LIN {X 0,Y 131.785,Z 325.121,A -85,B 0,C 180,E1 -26219.114,E2 -26219.114} C_VEL
LIN {X 0,Y 136.517,Z 312.595,A -85,B 0,C 180,E1 -26221.843,E2 -26221.843} C_VEL
LIN {X 0,Y 140.644,Z 299.524,A -85,B 0,C 180,E1 -26223.984,E2 -26223.984} C_VEL
LIN {X 0,Y 143.918,Z 286.061,A -85,B 0,C 180,E1 -26225.653,E2 -26225.653} C_VEL
LIN {X 0,Y 146.479,Z 272.18,A -85,B 0,C 180,E1 -26226.846,E2 -26226.846} C_VEL
LIN {X 0,Y 148.119,Z 259.286,A -85,B 0,C 180,E1 -26227.542,E2 -26227.542} C_VEL
LIN {X 0,Y 152.361,Z 207.8,A -85,B 0,C 180,E1 -26229.457,E2 -26229.457} C_VEL
LIN {X 0,Y 147.363,Z 196.9,A -85,B 0,C 180,E1 -26232.578,E2 -26232.578} C_VEL
LIN {X 0,Y 142.317,Z 187.434,A -85,B 0,C 180,E1 -26236.042,E2 -26236.042} C_VEL
LIN {X 0,Y 138.298,Z 180.817,A -85,B 0,C 180,E1 -26239.137,E2 -26239.137} C_VEL
LIN {X 0,Y 134.118,Z 174.322,A -85,B 0,C 180,E1 -26242.853,E2 -26242.853} C_VEL
LIN {X 0,Y 130.981,Z 169.962,A -85,B 0,C 180,E1 -26246.076,E2 -26246.076} C_VEL
LIN {X 0,Y 128.411,Z 166.477,A -85,B 0,C 180,E1 -26249.154,E2 -26249.154} C_VEL
LIN {X 0,Y 127.763,Z 165.521,A -85,B 0,C 180,E1 -26250.031,E2 -26250.031} C_VEL
LIN {X 0,Y 125.309,Z 162.834,A -85,B 0,C 180,E1 -26253.6,E2 -26253.6} C_VEL
LIN {X 0,Y 124.174,Z 160.568,A -85,B 0,C 180,E1 -26255.787,E2 -26255.787} C_VEL
LIN {X 0,Y 121.255,Z 158.023,A -85,B 0,C 180,E1 -26262.732,E2 -26262.732} C_VEL
LIN {X 0,Y 120.363,Z 155.046,A -85,B 0,C 180,E1 -26268.375,E2 -26268.375} C_VEL
LIN {X 0,Y 120.599,Z 154.855,A -85,B 0,C 180,E1 -26276.67,E2 -26276.67} C_VEL
LIN {X 0,Y 120.863,Z 155.058,A -85,B 0,C 180,E1 -26278.137,E2 -26278.137} C_VEL
LIN {X 0,Y 121.622,Z 157.801,A -85,B 0,C 180,E1 -26281.874,E2 -26281.874} C_VEL
LIN {X 0,Y 123.928,Z 160.174,A -85,B 0,C 180,E1 -26287.341,E2 -26287.341} C_VEL
LIN {X 0,Y 124.584,Z 160.744,A -85,B 0,C 180,E1 -26288.526,E2 -26288.526} C_VEL
LIN {X 0,Y 126.362,Z 163.972,A -85,B 0,C 180,E1 -26291.642,E2 -26291.642} C_VEL
LIN {X 0,Y 128.449,Z 166.176,A -85,B 0,C 180,E1 -26294.466,E2 -26294.466} C_VEL
LIN {X 0,Y 131.151,Z 169.964,A -85,B 0,C 180,E1 -26297.718,E2 -26297.718} C_VEL
LIN {X 0,Y 135.213,Z 176.102,A -85,B 0,C 180,E1 -26301.831,E2 -26301.831} C_VEL
LIN {X 0,Y 137.802,Z 180.05,A -85,B 0,C 180,E1 -26304.089,E2 -26304.089} C_VEL
LIN {X 0,Y 142.126,Z 187.185,A -85,B 0,C 180,E1 -26307.455,E2 -26307.455} C_VEL
LIN {X 0,Y 145.883,Z 194.238,A -85,B 0,C 180,E1 -26310.095,E2 -26310.095} C_VEL
LIN {X 0,Y 150.285,Z 206.436,A -85,B 0,C 180,E1 -26313.156,E2 -26313.156} C_VEL
LIN {X 0,Y 152.14,Z 212.6,A -85,B 0,C 180,E1 -26314.415,E2 -26314.415} C_VEL
LIN {X 0,Y 147.502,Z 269.5,A -85,B 0,C 180,E1 -26316.633,E2 -26316.633} C_VEL
LIN {X 0,Y 145.233,Z 284.149,A -85,B 0,C 180,E1 -26317.596,E2 -26317.596} C_VEL
LIN {X 0,Y 142.182,Z 297.577,A -85,B 0,C 180,E1 -26318.882,E2 -26318.882} C_VEL
LIN {X 0,Y 138.14,Z 311.67,A -85,B 0,C 180,E1 -26320.826,E2 -26320.826} C_VEL
LIN {X 0,Y 133.661,Z 324.178,A -85,B 0,C 180,E1 -26323.133,E2 -26323.133} C_VEL
LIN {X 0,Y 130.05,Z 333.38,A -85,B 0,C 180,E1 -26325.376,E2 -26325.376} C_VEL
LIN {X 0,Y 126.93,Z 340.175,A -85,B 0,C 180,E1 -26327.298,E2 -26327.298} C_VEL
LIN {X 0,Y 122.296,Z 349.988,A -85,B 0,C 180,E1 -26330.798,E2 -26330.798} C_VEL
LIN {X 0,Y 117.358,Z 359.79,A -85,B 0,C 180,E1 -26335.332,E2 -26335.332} C_VEL
LIN {X 0,Y 112.94,Z 368.47,A -85,B 0,C 180,E1 -26340.617,E2 -26340.617} C_VEL
LIN {X 0,Y 109.945,Z 374.628,A -85,B 0,C 180,E1 -26345.455,E2 -26345.455} C_VEL
LIN {X 0,Y 107.473,Z 380.188,A -85,B 0,C 180,E1 -26350.921,E2 -26350.921} C_VEL
LIN {X 0,Y 105.927,Z 384.738,A -85,B 0,C 180,E1 -26356.578,E2 -26356.578} C_VEL
LIN {X 0,Y 105.224,Z 388.285,A -85,B 0,C 180,E1 -26362.329,E2 -26362.329} C_VEL
LIN {X 0,Y 105.192,Z 391.7,A -85,B 0,C 180,E1 -26370.005,E2 -26370.005} C_VEL
LIN {X 0,Y 105.119,Z 392.843,A -85,B 0,C 180,E1 -26373.839,E2 -26373.839} C_VEL
LIN {X 0,Y 105.704,Z 394.109,A -85,B 0,C 180,E1 -26381.511,E2 -26381.511} C_VEL
LIN {X 0,Y 107.789,Z 394.075,A -85,B 0,C 180,E1 -26389.032,E2 -26389.032} C_VEL
LIN {X 0,Y 111.681,Z 392.762,A -85,B 0,C 180,E1 -26396.141,E2 -26396.141} C_VEL
LIN {X 0,Y 117.55,Z 389.878,A -85,B 0,C 180,E1 -26403.156,E2 -26403.156} C_VEL
LIN {X 0,Y 124.609,Z 385.666,A -85,B 0,C 180,E1 -26409.134,E2 -26409.134} C_VEL
LIN {X 0,Y 127.112,Z 383.711,A -85,B 0,C 180,E1 -26411.401,E2 -26411.401} C_VEL
LIN {X 0,Y 130.13,Z 380.239,A -85,B 0,C 180,E1 -26415.327,E2 -26415.327} C_VEL
LIN {X 0,Y 133.647,Z 376.305,A -85,B 0,C 180,E1 -26418.958,E2 -26418.958} C_VEL
LIN {X 0,Y 136.798,Z 373.53,A -85,B 0,C 180,E1 -26420.711,E2 -26420.711} C_VEL
LIN {X 0,Y 145.544,Z 366.023,A -85,B 0,C 180,E1 -26423.987,E2 -26423.987} C_VEL
LIN {X 0,Y 154.63,Z 356.799,A -85,B 0,C 180,E1 -26426.995,E2 -26426.995} C_VEL
LIN {X 0,Y 163.45,Z 346.525,A -85,B 0,C 180,E1 -26429.318,E2 -26429.318} C_VEL
LIN {X 0,Y 171.421,Z 335.451,A -85,B 0,C 180,E1 -26431.211,E2 -26431.211} C_VEL
LIN {X 0,Y 178.854,Z 323.08,A -85,B 0,C 180,E1 -26432.759,E2 -26432.759} C_VEL
LIN {X 0,Y 184.948,Z 310.841,A -85,B 0,C 180,E1 -26433.87,E2 -26433.87} C_VEL
LIN {X 0,Y 190.356,Z 297.238,A -85,B 0,C 180,E1 -26434.769,E2 -26434.769} C_VEL
LIN {X 0,Y 194.439,Z 283.649,A -85,B 0,C 180,E1 -26435.428,E2 -26435.428} C_VEL
LIN {X 0,Y 197.393,Z 269.461,A -85,B 0,C 180,E1 -26435.918,E2 -26435.918} C_VEL
LIN {X 0,Y 199.287,Z 253.75,A -85,B 0,C 180,E1 -26436.344,E2 -26436.344} C_VEL
LIN {X 0,Y 197.239,Z 247.184,A -85,B 0,C 180,E1 -26439.469,E2 -26439.469} C_VEL
LIN {X 0,Y 195.601,Z 242.329,A -85,B 0,C 180,E1 -26442.751,E2 -26442.751} C_VEL
LIN {X 0,Y 194.612,Z 239.828,A -85,B 0,C 180,E1 -26445.351,E2 -26445.351} C_VEL
LIN {X 0,Y 193.533,Z 236.708,A -85,B 0,C 180,E1 -26451.641,E2 -26451.641} C_VEL
LIN {X 0,Y 193.655,Z 236.699,A -85,B 0,C 180,E1 -26454.175,E2 -26454.175} C_VEL
LIN {X 0,Y 194.972,Z 240.283,A -85,B 0,C 180,E1 -26459.993,E2 -26459.993} C_VEL
LIN {X 0,Y 196.407,Z 243.777,A -85,B 0,C 180,E1 -26463.231,E2 -26463.231} C_VEL
LIN {X 0,Y 198.462,Z 248.413,A -85,B 0,C 180,E1 -26466.533,E2 -26466.533} C_VEL
LIN {X 0,Y 199.581,Z 251.089,A -85,B 0,C 180,E1 -26468.026,E2 -26468.026} C_VEL
LIN {X 0,Y 197.317,Z 268.586,A -85,B 0,C 180,E1 -26468.483,E2 -26468.483} C_VEL
LIN {X 0,Y 194.205,Z 282.706,A -85,B 0,C 180,E1 -26469.03,E2 -26469.03} C_VEL
LIN {X 0,Y 190.296,Z 295.309,A -85,B 0,C 180,E1 -26469.712,E2 -26469.712} C_VEL
LIN {X 0,Y 185.117,Z 308.406,A -85,B 0,C 180,E1 -26470.741,E2 -26470.741} C_VEL
LIN {X 0,Y 178.785,Z 321.148,A -85,B 0,C 180,E1 -26472.074,E2 -26472.074} C_VEL
LIN {X 0,Y 171.815,Z 332.614,A -85,B 0,C 180,E1 -26473.649,E2 -26473.649} C_VEL
LIN {X 0,Y 164.146,Z 343.198,A -85,B 0,C 180,E1 -26475.548,E2 -26475.548} C_VEL
LIN {X 0,Y 156.73,Z 352.032,A -85,B 0,C 180,E1 -26477.648,E2 -26477.648} C_VEL
LIN {X 0,Y 148.112,Z 360.829,A -85,B 0,C 180,E1 -26480.412,E2 -26480.412} C_VEL
LIN {X 0,Y 139.155,Z 368.672,A -85,B 0,C 180,E1 -26483.82,E2 -26483.82} C_VEL
LIN {X 0,Y 130.898,Z 374.913,A -85,B 0,C 180,E1 -26487.629,E2 -26487.629} C_VEL
LIN {X 0,Y 123.838,Z 379.589,A -85,B 0,C 180,E1 -26491.642,E2 -26491.642} C_VEL
LIN {X 0,Y 115.677,Z 384.073,A -85,B 0,C 180,E1 -26497.397,E2 -26497.397} C_VEL
LIN {X 0,Y 108.425,Z 387.236,A -85,B 0,C 180,E1 -26504.513,E2 -26504.513} C_VEL
LIN {X 0,Y 103.082,Z 388.764,A -85,B 0,C 180,E1 -26512.142,E2 -26512.142} C_VEL
LIN {X 0,Y 99.548,Z 388.842,A -85,B 0,C 180,E1 -26520.377,E2 -26520.377} C_VEL
LIN {X 0,Y 97.829,Z 387.459,A -85,B 0,C 180,E1 -26529.011,E2 -26529.011} C_VEL
LIN {X 0,Y 97.525,Z 386.246,A -85,B 0,C 180,E1 -26533.241,E2 -26533.241} C_VEL
LIN {X 0,Y 98.023,Z 382.697,A -85,B 0,C 180,E1 -26541.75,E2 -26541.75} C_VEL
LIN {X 0,Y 99.346,Z 379.08,A -85,B 0,C 180,E1 -26547.967,E2 -26547.967} C_VEL
LIN {X 0,Y 101.284,Z 374.503,A -85,B 0,C 180,E1 -26553.973,E2 -26553.973} C_VEL
LIN {X 0,Y 104.649,Z 367.913,A -85,B 0,C 180,E1 -26560.637,E2 -26560.637} C_VEL
LIN {X 0,Y 109.179,Z 359.737,A -85,B 0,C 180,E1 -26566.833,E2 -26566.833} C_VEL
LIN {X 0,Y 113.83,Z 351.181,A -85,B 0,C 180,E1 -26571.738,E2 -26571.738} C_VEL
LIN {X 0,Y 118.098,Z 342.71,A -85,B 0,C 180,E1 -26575.554,E2 -26575.554} C_VEL
LIN {X 0,Y 122.512,Z 333.725,A -85,B 0,C 180,E1 -26578.709,E2 -26578.709} C_VEL
LIN {X 0,Y 127.175,Z 323.103,A -85,B 0,C 180,E1 -26581.662,E2 -26581.662} C_VEL
LIN {X 0,Y 131.678,Z 311.646,A -85,B 0,C 180,E1 -26584.079,E2 -26584.079} C_VEL
LIN {X 0,Y 135.698,Z 299.286,A -85,B 0,C 180,E1 -26586.09,E2 -26586.09} C_VEL
LIN {X 0,Y 139.11,Z 285.7,A -85,B 0,C 180,E1 -26587.77,E2 -26587.77} C_VEL
LIN {X 0,Y 141.77,Z 271.607,A -85,B 0,C 180,E1 -26588.968,E2 -26588.968} C_VEL
LIN {X 0,Y 143.344,Z 259.679,A -85,B 0,C 180,E1 -26589.591,E2 -26589.591} C_VEL
LIN {X 0,Y 147.539,Z 210.291,A -85,B 0,C 180,E1 -26591.453,E2 -26591.453} C_VEL
LIN {X 0,Y 143.283,Z 200.805,A -85,B 0,C 180,E1 -26594.355,E2 -26594.355} C_VEL
LIN {X 0,Y 138.513,Z 191.636,A -85,B 0,C 180,E1 -26597.951,E2 -26597.951} C_VEL
LIN {X 0,Y 135.152,Z 185.928,A -85,B 0,C 180,E1 -26600.799,E2 -26600.799} C_VEL
LIN {X 0,Y 131.35,Z 179.866,A -85,B 0,C 180,E1 -26604.502,E2 -26604.502} C_VEL
LIN {X 0,Y 128.942,Z 176.298,A -85,B 0,C 180,E1 -26607.199,E2 -26607.199} C_VEL
LIN {X 0,Y 125.898,Z 171.998,A -85,B 0,C 180,E1 -26611.214,E2 -26611.214} C_VEL
LIN {X 0,Y 123.5,Z 168.944,A -85,B 0,C 180,E1 -26615.11,E2 -26615.11} C_VEL
LIN {X 0,Y 122.683,Z 167.345,A -85,B 0,C 180,E1 -26616.827,E2 -26616.827} C_VEL
LIN {X 0,Y 120.011,Z 164.606,A -85,B 0,C 180,E1 -26624.079,E2 -26624.079} C_VEL
LIN {X 0,Y 119.42,Z 162.041,A -85,B 0,C 180,E1 -26628.958,E2 -26628.958} C_VEL
LIN {X 0,Y 119.78,Z 161.905,A -85,B 0,C 180,E1 -26637.068,E2 -26637.068} C_VEL
LIN {X 0,Y 120.765,Z 165.154,A -85,B 0,C 180,E1 -26642.095,E2 -26642.095} C_VEL
LIN {X 0,Y 123.12,Z 167.53,A -85,B 0,C 180,E1 -26647.596,E2 -26647.596} C_VEL
LIN {X 0,Y 125.06,Z 170.939,A -85,B 0,C 180,E1 -26651.149,E2 -26651.149} C_VEL
LIN {X 0,Y 126.635,Z 172.708,A -85,B 0,C 180,E1 -26653.41,E2 -26653.41} C_VEL
LIN {X 0,Y 129.754,Z 177.467,A -85,B 0,C 180,E1 -26657.382,E2 -26657.382} C_VEL
LIN {X 0,Y 132.774,Z 182.144,A -85,B 0,C 180,E1 -26660.602,E2 -26660.602} C_VEL
LIN {X 0,Y 136.308,Z 187.774,A -85,B 0,C 180,E1 -26663.845,E2 -26663.845} C_VEL
LIN {X 0,Y 141.473,Z 197.254,A -85,B 0,C 180,E1 -26667.968,E2 -26667.968} C_VEL
LIN {X 0,Y 144.23,Z 204.494,A -85,B 0,C 180,E1 -26670.074,E2 -26670.074} C_VEL
LIN {X 0,Y 147.28,Z 214.262,A -85,B 0,C 180,E1 -26672.362,E2 -26672.362} C_VEL
LIN {X 0,Y 146.746,Z 222.337,A -85,B 0,C 180,E1 -26672.728,E2 -26672.728} C_VEL
LIN {X 0,Y 142.689,Z 269.498,A -85,B 0,C 180,E1 -26674.575,E2 -26674.575} C_VEL
LIN {X 0,Y 140.338,Z 284.088,A -85,B 0,C 180,E1 -26675.54,E2 -26675.54} C_VEL
LIN {X 0,Y 137.174,Z 297.482,A -85,B 0,C 180,E1 -26676.826,E2 -26676.826} C_VEL
LIN {X 0,Y 132.966,Z 311.555,A -85,B 0,C 180,E1 -26678.782,E2 -26678.782} C_VEL
LIN {X 0,Y 128.257,Z 324.129,A -85,B 0,C 180,E1 -26681.126,E2 -26681.126} C_VEL
LIN {X 0,Y 123.909,Z 334.415,A -85,B 0,C 180,E1 -26683.69,E2 -26683.69} C_VEL
LIN {X 0,Y 119.753,Z 343.17,A -85,B 0,C 180,E1 -26686.41,E2 -26686.41} C_VEL
LIN {X 0,Y 114.954,Z 352.479,A -85,B 0,C 180,E1 -26690.07,E2 -26690.07} C_VEL
LIN {X 0,Y 109.973,Z 361.805,A -85,B 0,C 180,E1 -26694.896,E2 -26694.896} C_VEL
LIN {X 0,Y 105.124,Z 370.633,A -85,B 0,C 180,E1 -26700.972,E2 -26700.972} C_VEL
LIN {X 0,Y 101.599,Z 377.833,A -85,B 0,C 180,E1 -26707.644,E2 -26707.644} C_VEL
LIN {X 0,Y 99.478,Z 382.767,A -85,B 0,C 180,E1 -26713.591,E2 -26713.591} C_VEL
LIN {X 0,Y 98.36,Z 386.753,A -85,B 0,C 180,E1 -26719.716,E2 -26719.716} C_VEL
LIN {X 0,Y 97.958,Z 389.767,A -85,B 0,C 180,E1 -26725.892,E2 -26725.892} C_VEL
LIN {X 0,Y 98.096,Z 391.33,A -85,B 0,C 180,E1 -26730.006,E2 -26730.006} C_VEL
LIN {X 0,Y 98.029,Z 392.512,A -85,B 0,C 180,E1 -26734.117,E2 -26734.117} C_VEL
LIN {X 0,Y 98.727,Z 393.855,A -85,B 0,C 180,E1 -26742.337,E2 -26742.337} C_VEL
LIN {X 0,Y 101.062,Z 393.897,A -85,B 0,C 180,E1 -26750.353,E2 -26750.353} C_VEL
LIN {X 0,Y 105.312,Z 392.666,A -85,B 0,C 180,E1 -26757.855,E2 -26757.855} C_VEL
LIN {X 0,Y 111.235,Z 390.106,A -85,B 0,C 180,E1 -26764.761,E2 -26764.761} C_VEL
LIN {X 0,Y 118.785,Z 386.017,A -85,B 0,C 180,E1 -26771.031,E2 -26771.031} C_VEL
LIN {X 0,Y 126.949,Z 380.85,A -85,B 0,C 180,E1 -26776.035,E2 -26776.035} C_VEL
LIN {X 0,Y 133.996,Z 375.737,A -85,B 0,C 180,E1 -26779.516,E2 -26779.516} C_VEL
LIN {X 0,Y 136.798,Z 373.53,A -85,B 0,C 180,E1 -26780.711,E2 -26780.711} C_VEL
LIN {X 0,Y 140.02,Z 370.6,A -85,B 0,C 180,E1 -26782.368,E2 -26782.368} C_VEL
LIN {X 0,Y 144.13,Z 365.612,A -85,B 0,C 180,E1 -26785.423,E2 -26785.423} C_VEL
LIN {X 0,Y 148.392,Z 360.229,A -85,B 0,C 180,E1 -26788.22,E2 -26788.22} C_VEL
LIN {X 0,Y 151.719,Z 356.527,A -85,B 0,C 180,E1 -26789.455,E2 -26789.455} C_VEL
LIN {X 0,Y 159.972,Z 347.234,A -85,B 0,C 180,E1 -26791.487,E2 -26791.487} C_VEL
LIN {X 0,Y 168.149,Z 336.362,A -85,B 0,C 180,E1 -26793.31,E2 -26793.31} C_VEL
LIN {X 0,Y 175.75,Z 324.317,A -85,B 0,C 180,E1 -26794.795,E2 -26794.795} C_VEL
LIN {X 0,Y 181.969,Z 312.422,A -85,B 0,C 180,E1 -26795.852,E2 -26795.852} C_VEL
LIN {X 0,Y 187.479,Z 299.317,A -85,B 0,C 180,E1 -26796.704,E2 -26796.704} C_VEL
LIN {X 0,Y 191.819,Z 285.809,A -85,B 0,C 180,E1 -26797.36,E2 -26797.36} C_VEL
LIN {X 0,Y 195.027,Z 271.716,A -85,B 0,C 180,E1 -26797.841,E2 -26797.841} C_VEL
LIN {X 0,Y 196.958,Z 257.662,A -85,B 0,C 180,E1 -26798.223,E2 -26798.223} C_VEL
LIN {X 0,Y 195.511,Z 252.638,A -85,B 0,C 180,E1 -26800.84,E2 -26800.84} C_VEL
LIN {X 0,Y 194.366,Z 248.965,A -85,B 0,C 180,E1 -26803.45,E2 -26803.45} C_VEL
LIN {X 0,Y 193.551,Z 246.75,A -85,B 0,C 180,E1 -26805.806,E2 -26805.806} C_VEL
LIN {X 0,Y 192.64,Z 243.839,A -85,B 0,C 180,E1 -26811.602,E2 -26811.602} C_VEL
LIN {X 0,Y 192.762,Z 243.785,A -85,B 0,C 180,E1 -26814.148,E2 -26814.148} C_VEL
LIN {X 0,Y 193.91,Z 247.232,A -85,B 0,C 180,E1 -26819.604,E2 -26819.604} C_VEL
LIN {X 0,Y 195.252,Z 250.712,A -85,B 0,C 180,E1 -26822.83,E2 -26822.83} C_VEL
LIN {X 0,Y 197.001,Z 254.991,A -85,B 0,C 180,E1 -26825.861,E2 -26825.861} C_VEL
LIN {X 0,Y 197.173,Z 255.515,A -85,B 0,C 180,E1 -26826.131,E2 -26826.131} C_VEL
LIN {X 0,Y 194.888,Z 271.324,A -85,B 0,C 180,E1 -26826.569,E2 -26826.569} C_VEL
LIN {X 0,Y 191.611,Z 284.922,A -85,B 0,C 180,E1 -26827.096,E2 -26827.096} C_VEL
LIN {X 0,Y 187.538,Z 297.332,A -85,B 0,C 180,E1 -26827.78,E2 -26827.78} C_VEL
LIN {X 0,Y 182.006,Z 310.472,A -85,B 0,C 180,E1 -26828.803,E2 -26828.803} C_VEL
LIN {X 0,Y 175.763,Z 322.402,A -85,B 0,C 180,E1 -26830.037,E2 -26830.037} C_VEL
LIN {X 0,Y 168.582,Z 333.724,A -85,B 0,C 180,E1 -26831.552,E2 -26831.552} C_VEL
LIN {X 0,Y 160.745,Z 344.114,A -85,B 0,C 180,E1 -26833.38,E2 -26833.38} C_VEL
LIN {X 0,Y 153.106,Z 352.829,A -85,B 0,C 180,E1 -26835.416,E2 -26835.416} C_VEL
LIN {X 0,Y 144.203,Z 361.522,A -85,B 0,C 180,E1 -26838.116,E2 -26838.116} C_VEL
LIN {X 0,Y 135.242,Z 369.009,A -85,B 0,C 180,E1 -26841.32,E2 -26841.32} C_VEL
LIN {X 0,Y 127.563,Z 374.594,A -85,B 0,C 180,E1 -26844.615,E2 -26844.615} C_VEL
LIN {X 0,Y 120.034,Z 379.342,A -85,B 0,C 180,E1 -26848.558,E2 -26848.558} C_VEL
LIN {X 0,Y 113.068,Z 383.068,A -85,B 0,C 180,E1 -26852.944,E2 -26852.944} C_VEL
LIN {X 0,Y 106.875,Z 385.886,A -85,B 0,C 180,E1 -26857.889,E2 -26857.889} C_VEL
LIN {X 0,Y 99.994,Z 388.261,A -85,B 0,C 180,E1 -26865.337,E2 -26865.337} C_VEL
LIN {X 0,Y 94.911,Z 389.164,A -85,B 0,C 180,E1 -26873.666,E2 -26873.666} C_VEL
LIN {X 0,Y 91.732,Z 388.629,A -85,B 0,C 180,E1 -26882.626,E2 -26882.626} C_VEL
LIN {X 0,Y 90.783,Z 387.614,A -85,B 0,C 180,E1 -26888.233,E2 -26888.233} C_VEL
LIN {X 0,Y 90.401,Z 385.149,A -85,B 0,C 180,E1 -26896.506,E2 -26896.506} C_VEL
LIN {X 0,Y 91.628,Z 380.96,A -85,B 0,C 180,E1 -26905.595,E2 -26905.595} C_VEL
LIN {X 0,Y 93.362,Z 376.841,A -85,B 0,C 180,E1 -26912.151,E2 -26912.151} C_VEL
LIN {X 0,Y 95.921,Z 371.716,A -85,B 0,C 180,E1 -26918.42,E2 -26918.42} C_VEL
LIN {X 0,Y 100.204,Z 364.386,A -85,B 0,C 180,E1 -26925.243,E2 -26925.243} C_VEL
LIN {X 0,Y 105.04,Z 356.234,A -85,B 0,C 180,E1 -26930.915,E2 -26930.915} C_VEL
LIN {X 0,Y 109.98,Z 347.504,A -85,B 0,C 180,E1 -26935.547,E2 -26935.547} C_VEL
LIN {X 0,Y 115.154,Z 337.389,A -85,B 0,C 180,E1 -26939.722,E2 -26939.722} C_VEL
LIN {X 0,Y 120.652,Z 326.189,A -85,B 0,C 180,E1 -26943.094,E2 -26943.094} C_VEL
LIN {X 0,Y 125.837,Z 313.828,A -85,B 0,C 180,E1 -26945.898,E2 -26945.898} C_VEL
LIN {X 0,Y 130.004,Z 301.967,A -85,B 0,C 180,E1 -26947.941,E2 -26947.941} C_VEL
LIN {X 0,Y 133.573,Z 289.115,A -85,B 0,C 180,E1 -26949.634,E2 -26949.634} C_VEL
LIN {X 0,Y 136.656,Z 274.476,A -85,B 0,C 180,E1 -26950.968,E2 -26950.968} C_VEL
LIN {X 0,Y 138.496,Z 261.774,A -85,B 0,C 180,E1 -26951.721,E2 -26951.721} C_VEL
LIN {X 0,Y 142.916,Z 212.87,A -85,B 0,C 180,E1 -26953.544,E2 -26953.544} C_VEL
LIN {X 0,Y 138.94,Z 203.896,A -85,B 0,C 180,E1 -26956.546,E2 -26956.546} C_VEL
LIN {X 0,Y 134.376,Z 194.924,A -85,B 0,C 180,E1 -26960.411,E2 -26960.411} C_VEL
LIN {X 0,Y 129.944,Z 187.265,A -85,B 0,C 180,E1 -26964.826,E2 -26964.826} C_VEL
LIN {X 0,Y 126.936,Z 182.619,A -85,B 0,C 180,E1 -26968.378,E2 -26968.378} C_VEL
LIN {X 0,Y 124.256,Z 178.611,A -85,B 0,C 180,E1 -26972.186,E2 -26972.186} C_VEL
LIN {X 0,Y 121.836,Z 175.161,A -85,B 0,C 180,E1 -26976.527,E2 -26976.527} C_VEL
LIN {X 0,Y 121.406,Z 174.223,A -85,B 0,C 180,E1 -26977.53,E2 -26977.53} C_VEL
LIN {X 0,Y 118.84,Z 171.148,A -85,B 0,C 180,E1 -26985.455,E2 -26985.455} C_VEL
LIN {X 0,Y 118.483,Z 168.952,A -85,B 0,C 180,E1 -26989.761,E2 -26989.761} C_VEL
LIN {X 0,Y 118.825,Z 169.057,A -85,B 0,C 180,E1 -26996.774,E2 -26996.774} C_VEL
LIN {X 0,Y 119.66,Z 172.036,A -85,B 0,C 180,E1 -27001.464,E2 -27001.464} C_VEL
LIN {X 0,Y 121.74,Z 174.355,A -85,B 0,C 180,E1 -27006.745,E2 -27006.745} C_VEL
LIN {X 0,Y 123.649,Z 177.74,A -85,B 0,C 180,E1 -27010.449,E2 -27010.449} C_VEL
LIN {X 0,Y 125.043,Z 179.504,A -85,B 0,C 180,E1 -27012.59,E2 -27012.59} C_VEL
LIN {X 0,Y 127.779,Z 183.879,A -85,B 0,C 180,E1 -27016.309,E2 -27016.309} C_VEL
LIN {X 0,Y 130.599,Z 188.472,A -85,B 0,C 180,E1 -27019.536,E2 -27019.536} C_VEL
LIN {X 0,Y 133.937,Z 194.178,A -85,B 0,C 180,E1 -27022.826,E2 -27022.826} C_VEL
LIN {X 0,Y 138.497,Z 203.038,A -85,B 0,C 180,E1 -27026.738,E2 -27026.738} C_VEL
LIN {X 0,Y 142.194,Z 214.449,A -85,B 0,C 180,E1 -27029.833,E2 -27029.833} C_VEL
LIN {X 0,Y 142.782,Z 216.469,A -85,B 0,C 180,E1 -27030.308,E2 -27030.308} C_VEL
LIN {X 0,Y 138.047,Z 269.577,A -85,B 0,C 180,E1 -27032.389,E2 -27032.389} C_VEL
LIN {X 0,Y 135.715,Z 283.578,A -85,B 0,C 180,E1 -27033.308,E2 -27033.308} C_VEL
LIN {X 0,Y 132.354,Z 297.333,A -85,B 0,C 180,E1 -27034.617,E2 -27034.617} C_VEL
LIN {X 0,Y 128.594,Z 309.614,A -85,B 0,C 180,E1 -27036.289,E2 -27036.289} C_VEL
LIN {X 0,Y 123.442,Z 323.025,A -85,B 0,C 180,E1 -27038.722,E2 -27038.722} C_VEL
LIN {X 0,Y 119.117,Z 333.081,A -85,B 0,C 180,E1 -27041.221,E2 -27041.221} C_VEL
LIN {X 0,Y 115.167,Z 340.96,A -85,B 0,C 180,E1 -27043.567,E2 -27043.567} C_VEL
LIN {X 0,Y 109.55,Z 351.477,A -85,B 0,C 180,E1 -27047.661,E2 -27047.661} C_VEL
LIN {X 0,Y 104.168,Z 360.949,A -85,B 0,C 180,E1 -27052.619,E2 -27052.619} C_VEL
LIN {X 0,Y 99.202,Z 369.361,A -85,B 0,C 180,E1 -27058.501,E2 -27058.501} C_VEL
LIN {X 0,Y 95.955,Z 375.307,A -85,B 0,C 180,E1 -27063.938,E2 -27063.938} C_VEL
LIN {X 0,Y 93.279,Z 380.654,A -85,B 0,C 180,E1 -27070.188,E2 -27070.188} C_VEL
LIN {X 0,Y 91.354,Z 386.266,A -85,B 0,C 180,E1 -27078.918,E2 -27078.918} C_VEL
LIN {X 0,Y 90.886,Z 389.358,A -85,B 0,C 180,E1 -27085.571,E2 -27085.571} C_VEL
LIN {X 0,Y 90.993,Z 390.961,A -85,B 0,C 180,E1 -27090.006,E2 -27090.006} C_VEL
LIN {X 0,Y 90.936,Z 392.18,A -85,B 0,C 180,E1 -27094.439,E2 -27094.439} C_VEL
LIN {X 0,Y 91.783,Z 393.599,A -85,B 0,C 180,E1 -27103.287,E2 -27103.287} C_VEL
LIN {X 0,Y 94.396,Z 393.721,A -85,B 0,C 180,E1 -27111.862,E2 -27111.862} C_VEL
LIN {X 0,Y 99.051,Z 392.572,A -85,B 0,C 180,E1 -27119.787,E2 -27119.787} C_VEL
LIN {X 0,Y 105.375,Z 390.129,A -85,B 0,C 180,E1 -27126.895,E2 -27126.895} C_VEL
LIN {X 0,Y 113.114,Z 386.332,A -85,B 0,C 180,E1 -27133.121,E2 -27133.121} C_VEL
LIN {X 0,Y 122.11,Z 381.063,A -85,B 0,C 180,E1 -27138.442,E2 -27138.442} C_VEL
LIN {X 0,Y 129.499,Z 376.004,A -85,B 0,C 180,E1 -27141.906,E2 -27141.906} C_VEL
LIN {X 0,Y 138.766,Z 368.815,A -85,B 0,C 180,E1 -27145.394,E2 -27145.394} C_VEL
LIN {X 0,Y 147.442,Z 360.885,A -85,B 0,C 180,E1 -27148.223,E2 -27148.223} C_VEL
LIN {X 0,Y 151.719,Z 356.527,A -85,B 0,C 180,E1 -27149.455,E2 -27149.455} C_VEL
LIN {X 0,Y 155.057,Z 352.734,A -85,B 0,C 180,E1 -27150.608,E2 -27150.608} C_VEL
LIN {X 0,Y 159.471,Z 346.422,A -85,B 0,C 180,E1 -27152.898,E2 -27152.898} C_VEL
LIN {X 0,Y 163.706,Z 339.638,A -85,B 0,C 180,E1 -27154.972,E2 -27154.972} C_VEL
LIN {X 0,Y 166.651,Z 335.11,A -85,B 0,C 180,E1 -27155.792,E2 -27155.792} C_VEL
LIN {X 0,Y 174.458,Z 322.752,A -85,B 0,C 180,E1 -27157.156,E2 -27157.156} C_VEL
LIN {X 0,Y 180.784,Z 310.541,A -85,B 0,C 180,E1 -27158.155,E2 -27158.155} C_VEL
LIN {X 0,Y 186.401,Z 296.966,A -85,B 0,C 180,E1 -27158.941,E2 -27158.941} C_VEL
LIN {X 0,Y 190.783,Z 283.007,A -85,B 0,C 180,E1 -27159.5,E2 -27159.5} C_VEL
LIN {X 0,Y 193.817,Z 268.809,A -85,B 0,C 180,E1 -27159.959,E2 -27159.959} C_VEL
LIN {X 0,Y 194.819,Z 261.782,A -85,B 0,C 180,E1 -27160.143,E2 -27160.143} C_VEL
LIN {X 0,Y 193.961,Z 258.48,A -85,B 0,C 180,E1 -27162.055,E2 -27162.055} C_VEL
LIN {X 0,Y 193.163,Z 255.576,A -85,B 0,C 180,E1 -27164.158,E2 -27164.158} C_VEL
LIN {X 0,Y 192.508,Z 253.629,A -85,B 0,C 180,E1 -27166.266,E2 -27166.266} C_VEL
LIN {X 0,Y 191.748,Z 250.817,A -85,B 0,C 180,E1 -27172.079,E2 -27172.079} C_VEL
LIN {X 0,Y 191.865,Z 250.893,A -85,B 0,C 180,E1 -27174.121,E2 -27174.121} C_VEL
LIN {X 0,Y 192.861,Z 254.147,A -85,B 0,C 180,E1 -27179.21,E2 -27179.21} C_VEL
LIN {X 0,Y 193.944,Z 257.216,A -85,B 0,C 180,E1 -27182.07,E2 -27182.07} C_VEL
LIN {X 0,Y 194.983,Z 260.105,A -85,B 0,C 180,E1 -27184.224,E2 -27184.224} C_VEL
LIN {X 0,Y 192.475,Z 274.658,A -85,B 0,C 180,E1 -27184.643,E2 -27184.643} C_VEL
LIN {X 0,Y 188.71,Z 288.649,A -85,B 0,C 180,E1 -27185.187,E2 -27185.187} C_VEL
LIN {X 0,Y 183.738,Z 302.29,A -85,B 0,C 180,E1 -27185.985,E2 -27185.985} C_VEL
LIN {X 0,Y 177.759,Z 315.151,A -85,B 0,C 180,E1 -27187.05,E2 -27187.05} C_VEL
LIN {X 0,Y 170.505,Z 327.639,A -85,B 0,C 180,E1 -27188.389,E2 -27188.389} C_VEL
LIN {X 0,Y 162.901,Z 338.465,A -85,B 0,C 180,E1 -27189.929,E2 -27189.929} C_VEL
LIN {X 0,Y 154.404,Z 348.649,A -85,B 0,C 180,E1 -27191.854,E2 -27191.854} C_VEL
LIN {X 0,Y 145.097,Z 358.129,A -85,B 0,C 180,E1 -27194.351,E2 -27194.351} C_VEL
LIN {X 0,Y 136.048,Z 365.924,A -85,B 0,C 180,E1 -27197.109,E2 -27197.109} C_VEL
LIN {X 0,Y 127.392,Z 372.351,A -85,B 0,C 180,E1 -27200.293,E2 -27200.293} C_VEL
LIN {X 0,Y 117.713,Z 378.444,A -85,B 0,C 180,E1 -27204.691,E2 -27204.691} C_VEL
LIN {X 0,Y 109.13,Z 382.928,A -85,B 0,C 180,E1 -27209.601,E2 -27209.601} C_VEL
LIN {X 0,Y 102.383,Z 385.857,A -85,B 0,C 180,E1 -27214.53,E2 -27214.53} C_VEL
LIN {X 0,Y 94.746,Z 388.338,A -85,B 0,C 180,E1 -27222.108,E2 -27222.108} C_VEL
LIN {X 0,Y 88.916,Z 389.346,A -85,B 0,C 180,E1 -27230.77,E2 -27230.77} C_VEL
LIN {X 0,Y 85.122,Z 388.914,A -85,B 0,C 180,E1 -27240.297,E2 -27240.297} C_VEL
LIN {X 0,Y 83.796,Z 387.781,A -85,B 0,C 180,E1 -27247.26,E2 -27247.26} C_VEL
LIN {X 0,Y 83.261,Z 385.595,A -85,B 0,C 180,E1 -27255.324,E2 -27255.324} C_VEL
LIN {X 0,Y 83.914,Z 382.677,A -85,B 0,C 180,E1 -27262.776,E2 -27262.776} C_VEL
LIN {X 0,Y 85.491,Z 378.934,A -85,B 0,C 180,E1 -27269.993,E2 -27269.993} C_VEL
LIN {X 0,Y 87.85,Z 374.278,A -85,B 0,C 180,E1 -27276.886,E2 -27276.886} C_VEL
LIN {X 0,Y 91.896,Z 367.526,A -85,B 0,C 180,E1 -27284.385,E2 -27284.385} C_VEL
LIN {X 0,Y 97.257,Z 359.105,A -85,B 0,C 180,E1 -27291.174,E2 -27291.174} C_VEL
LIN {X 0,Y 102.664,Z 350.288,A -85,B 0,C 180,E1 -27296.447,E2 -27296.447} C_VEL
LIN {X 0,Y 108.485,Z 339.763,A -85,B 0,C 180,E1 -27301.209,E2 -27301.209} C_VEL
LIN {X 0,Y 114.23,Z 328.993,A -85,B 0,C 180,E1 -27304.682,E2 -27304.682} C_VEL
LIN {X 0,Y 119.5,Z 317.291,A -85,B 0,C 180,E1 -27307.596,E2 -27307.596} C_VEL
LIN {X 0,Y 123.845,Z 306.158,A -85,B 0,C 180,E1 -27309.668,E2 -27309.668} C_VEL
LIN {X 0,Y 128.204,Z 292.17,A -85,B 0,C 180,E1 -27311.651,E2 -27311.651} C_VEL
LIN {X 0,Y 131.525,Z 278.055,A -85,B 0,C 180,E1 -27313.069,E2 -27313.069} C_VEL
LIN {X 0,Y 133.858,Z 263.75,A -85,B 0,C 180,E1 -27313.998,E2 -27313.998} C_VEL
LIN {X 0,Y 138.499,Z 215.692,A -85,B 0,C 180,E1 -27315.737,E2 -27315.737} C_VEL
LIN {X 0,Y 134.575,Z 206.557,A -85,B 0,C 180,E1 -27319.075,E2 -27319.075} C_VEL
LIN {X 0,Y 130.738,Z 198.829,A -85,B 0,C 180,E1 -27322.758,E2 -27322.758} C_VEL
LIN {X 0,Y 126.925,Z 192.104,A -85,B 0,C 180,E1 -27327.045,E2 -27327.045} C_VEL
LIN {X 0,Y 124.835,Z 188.728,A -85,B 0,C 180,E1 -27329.801,E2 -27329.801} C_VEL
LIN {X 0,Y 122.643,Z 185.192,A -85,B 0,C 180,E1 -27333.2,E2 -27333.2} C_VEL
LIN {X 0,Y 120.394,Z 181.745,A -85,B 0,C 180,E1 -27337.599,E2 -27337.599} C_VEL
LIN {X 0,Y 119.969,Z 180.957,A -85,B 0,C 180,E1 -27338.65,E2 -27338.65} C_VEL
LIN {X 0,Y 117.766,Z 177.789,A -85,B 0,C 180,E1 -27346.628,E2 -27346.628} C_VEL
LIN {X 0,Y 117.576,Z 175.964,A -85,B 0,C 180,E1 -27350.165,E2 -27350.165} C_VEL
LIN {X 0,Y 117.838,Z 176.044,A -85,B 0,C 180,E1 -27356.112,E2 -27356.112} C_VEL
LIN {X 0,Y 118.657,Z 179.065,A -85,B 0,C 180,E1 -27361.148,E2 -27361.148} C_VEL
LIN {X 0,Y 120.35,Z 181.121,A -85,B 0,C 180,E1 -27365.787,E2 -27365.787} C_VEL
LIN {X 0,Y 122.373,Z 184.668,A -85,B 0,C 180,E1 -27369.932,E2 -27369.932} C_VEL
LIN {X 0,Y 123.513,Z 186.359,A -85,B 0,C 180,E1 -27371.81,E2 -27371.81} C_VEL
LIN {X 0,Y 125.806,Z 190.193,A -85,B 0,C 180,E1 -27375.139,E2 -27375.139} C_VEL
LIN {X 0,Y 129.328,Z 196.282,A -85,B 0,C 180,E1 -27379.387,E2 -27379.387} C_VEL
LIN {X 0,Y 132.888,Z 203.17,A -85,B 0,C 180,E1 -27383.016,E2 -27383.016} C_VEL
LIN {X 0,Y 135.32,Z 208.531,A -85,B 0,C 180,E1 -27385.252,E2 -27385.252} C_VEL
LIN {X 0,Y 138.337,Z 218.52,A -85,B 0,C 180,E1 -27388.05,E2 -27388.05} C_VEL
LIN {X 0,Y 133.608,Z 269.568,A -85,B 0,C 180,E1 -27390.061,E2 -27390.061} C_VEL
LIN {X 0,Y 131.14,Z 283.674,A -85,B 0,C 180,E1 -27390.976,E2 -27390.976} C_VEL
LIN {X 0,Y 127.747,Z 297.086,A -85,B 0,C 180,E1 -27392.245,E2 -27392.245} C_VEL
LIN {X 0,Y 123.184,Z 311.168,A -85,B 0,C 180,E1 -27394.19,E2 -27394.19} C_VEL
LIN {X 0,Y 117.905,Z 324.071,A -85,B 0,C 180,E1 -27396.602,E2 -27396.602} C_VEL
LIN {X 0,Y 113.276,Z 334.036,A -85,B 0,C 180,E1 -27399.155,E2 -27399.155} C_VEL
LIN {X 0,Y 108.669,Z 342.79,A -85,B 0,C 180,E1 -27401.957,E2 -27401.957} C_VEL
LIN {X 0,Y 103.327,Z 352.104,A -85,B 0,C 180,E1 -27405.807,E2 -27405.807} C_VEL
LIN {X 0,Y 97.66,Z 361.428,A -85,B 0,C 180,E1 -27410.981,E2 -27410.981} C_VEL
LIN {X 0,Y 92.73,Z 369.234,A -85,B 0,C 180,E1 -27416.759,E2 -27416.759} C_VEL
LIN {X 0,Y 89.562,Z 374.592,A -85,B 0,C 180,E1 -27421.919,E2 -27421.919} C_VEL
LIN {X 0,Y 86.591,Z 380.046,A -85,B 0,C 180,E1 -27428.585,E2 -27428.585} C_VEL
LIN {X 0,Y 84.346,Z 385.753,A -85,B 0,C 180,E1 -27437.984,E2 -27437.984} C_VEL
LIN {X 0,Y 83.801,Z 388.936,A -85,B 0,C 180,E1 -27445.196,E2 -27445.196} C_VEL
LIN {X 0,Y 83.9,Z 390.581,A -85,B 0,C 180,E1 -27450.007,E2 -27450.007} C_VEL
LIN {X 0,Y 83.867,Z 391.841,A -85,B 0,C 180,E1 -27454.814,E2 -27454.814} C_VEL
LIN {X 0,Y 84.863,Z 393.34,A -85,B 0,C 180,E1 -27464.392,E2 -27464.392} C_VEL
LIN {X 0,Y 87.809,Z 393.544,A -85,B 0,C 180,E1 -27473.597,E2 -27473.597} C_VEL
LIN {X 0,Y 92.922,Z 392.478,A -85,B 0,C 180,E1 -27481.974,E2 -27481.974} C_VEL
LIN {X 0,Y 99.758,Z 390.119,A -85,B 0,C 180,E1 -27489.357,E2 -27489.357} C_VEL
LIN {X 0,Y 108.015,Z 386.409,A -85,B 0,C 180,E1 -27495.709,E2 -27495.709} C_VEL
LIN {X 0,Y 117.503,Z 381.242,A -85,B 0,C 180,E1 -27501.044,E2 -27501.044} C_VEL
LIN {X 0,Y 125.245,Z 376.271,A -85,B 0,C 180,E1 -27504.461,E2 -27504.461} C_VEL
LIN {X 0,Y 134.868,Z 369.189,A -85,B 0,C 180,E1 -27507.871,E2 -27507.871} C_VEL
LIN {X 0,Y 143.614,Z 361.587,A -85,B 0,C 180,E1 -27510.561,E2 -27510.561} C_VEL
LIN {X 0,Y 152.174,Z 353.016,A -85,B 0,C 180,E1 -27512.761,E2 -27512.761} C_VEL
LIN {X 0,Y 161.263,Z 342.372,A -85,B 0,C 180,E1 -27514.738,E2 -27514.738} C_VEL
LIN {X 0,Y 166.651,Z 335.11,A -85,B 0,C 180,E1 -27515.792,E2 -27515.792} C_VEL
LIN {X 0,Y 169.532,Z 330.521,A -85,B 0,C 180,E1 -27516.558,E2 -27516.558} C_VEL
LIN {X 0,Y 173.425,Z 322.878,A -85,B 0,C 180,E1 -27518.266,E2 -27518.266} C_VEL
LIN {X 0,Y 177.038,Z 315.005,A -85,B 0,C 180,E1 -27519.835,E2 -27519.835} C_VEL
LIN {X 0,Y 179.386,Z 309.884,A -85,B 0,C 180,E1 -27520.393,E2 -27520.393} C_VEL
LIN {X 0,Y 185.228,Z 295.858,A -85,B 0,C 180,E1 -27521.127,E2 -27521.127} C_VEL
LIN {X 0,Y 189.567,Z 281.988,A -85,B 0,C 180,E1 -27521.624,E2 -27521.624} C_VEL
LIN {X 0,Y 192.562,Z 267.873,A -85,B 0,C 180,E1 -27522.051,E2 -27522.051} C_VEL
LIN {X 0,Y 192.822,Z 265.827,A -85,B 0,C 180,E1 -27522.188,E2 -27522.188} C_VEL
LIN {X 0,Y 191.951,Z 262.175,A -85,B 0,C 180,E1 -27524.872,E2 -27524.872} C_VEL
LIN {X 0,Y 191.469,Z 260.525,A -85,B 0,C 180,E1 -27526.731,E2 -27526.731} C_VEL
LIN {X 0,Y 190.873,Z 257.786,A -85,B 0,C 180,E1 -27532.504,E2 -27532.504} C_VEL
LIN {X 0,Y 190.958,Z 257.882,A -85,B 0,C 180,E1 -27533.874,E2 -27533.874} C_VEL
LIN {X 0,Y 191.777,Z 261.047,A -85,B 0,C 180,E1 -27538.812,E2 -27538.812} C_VEL
LIN {X 0,Y 192.608,Z 263.857,A -85,B 0,C 180,E1 -27541.431,E2 -27541.431} C_VEL
LIN {X 0,Y 192.935,Z 264.866,A -85,B 0,C 180,E1 -27542.253,E2 -27542.253} C_VEL
LIN {X 0,Y 189.977,Z 279.286,A -85,B 0,C 180,E1 -27542.709,E2 -27542.709} C_VEL
LIN {X 0,Y 185.707,Z 293.241,A -85,B 0,C 180,E1 -27543.276,E2 -27543.276} C_VEL
LIN {X 0,Y 180.67,Z 305.813,A -85,B 0,C 180,E1 -27544.051,E2 -27544.051} C_VEL
LIN {X 0,Y 174.627,Z 317.845,A -85,B 0,C 180,E1 -27545.041,E2 -27545.041} C_VEL
LIN {X 0,Y 167.068,Z 330.064,A -85,B 0,C 180,E1 -27546.344,E2 -27546.344} C_VEL
LIN {X 0,Y 158.59,Z 341.369,A -85,B 0,C 180,E1 -27547.945,E2 -27547.945} C_VEL
LIN {X 0,Y 149.802,Z 351.204,A -85,B 0,C 180,E1 -27549.843,E2 -27549.843} C_VEL
LIN {X 0,Y 140.263,Z 360.284,A -85,B 0,C 180,E1 -27552.277,E2 -27552.277} C_VEL
LIN {X 0,Y 130.973,Z 367.734,A -85,B 0,C 180,E1 -27554.994,E2 -27554.994} C_VEL
LIN {X 0,Y 122.039,Z 373.85,A -85,B 0,C 180,E1 -27558.143,E2 -27558.143} C_VEL
LIN {X 0,Y 113.555,Z 378.826,A -85,B 0,C 180,E1 -27561.807,E2 -27561.807} C_VEL
LIN {X 0,Y 105.6,Z 382.788,A -85,B 0,C 180,E1 -27566.031,E2 -27566.031} C_VEL
LIN {X 0,Y 98.278,Z 385.795,A -85,B 0,C 180,E1 -27570.881,E2 -27570.881} C_VEL
LIN {X 0,Y 89.832,Z 388.416,A -85,B 0,C 180,E1 -27578.514,E2 -27578.514} C_VEL
LIN {X 0,Y 83.196,Z 389.528,A -85,B 0,C 180,E1 -27587.475,E2 -27587.475} C_VEL
LIN {X 0,Y 78.671,Z 389.198,A -85,B 0,C 180,E1 -27597.58,E2 -27597.58} C_VEL
LIN {X 0,Y 76.533,Z 387.436,A -85,B 0,C 180,E1 -27608.442,E2 -27608.442} C_VEL
LIN {X 0,Y 76.349,Z 384.255,A -85,B 0,C 180,E1 -27619.384,E2 -27619.384} C_VEL
LIN {X 0,Y 77.436,Z 381.353,A -85,B 0,C 180,E1 -27626.383,E2 -27626.383} C_VEL
LIN {X 0,Y 79.815,Z 376.613,A -85,B 0,C 180,E1 -27635.044,E2 -27635.044} C_VEL
LIN {X 0,Y 83.627,Z 370.394,A -85,B 0,C 180,E1 -27643.355,E2 -27643.355} C_VEL
LIN {X 0,Y 88.885,Z 362.63,A -85,B 0,C 180,E1 -27650.836,E2 -27650.836} C_VEL
LIN {X 0,Y 94.324,Z 354.537,A -85,B 0,C 180,E1 -27656.548,E2 -27656.548} C_VEL
LIN {X 0,Y 100.348,Z 344.81,A -85,B 0,C 180,E1 -27661.68,E2 -27661.68} C_VEL
LIN {X 0,Y 106.009,Z 335.058,A -85,B 0,C 180,E1 -27665.45,E2 -27665.45} C_VEL
LIN {X 0,Y 111.403,Z 324.585,A -85,B 0,C 180,E1 -27668.527,E2 -27668.527} C_VEL
LIN {X 0,Y 117.206,Z 311.724,A -85,B 0,C 180,E1 -27671.262,E2 -27671.262} C_VEL
LIN {X 0,Y 121.733,Z 299.254,A -85,B 0,C 180,E1 -27673.274,E2 -27673.274} C_VEL
LIN {X 0,Y 125.299,Z 286.758,A -85,B 0,C 180,E1 -27674.793,E2 -27674.793} C_VEL
LIN {X 0,Y 128.101,Z 274.053,A -85,B 0,C 180,E1 -27675.862,E2 -27675.862} C_VEL
LIN {X 0,Y 130.042,Z 261.256,A -85,B 0,C 180,E1 -27676.574,E2 -27676.574} C_VEL
LIN {X 0,Y 134.183,Z 218.974,A -85,B 0,C 180,E1 -27678.099,E2 -27678.099} C_VEL
LIN {X 0,Y 134.069,Z 217.826,A -85,B 0,C 180,E1 -27678.288,E2 -27678.288} C_VEL
LIN {X 0,Y 130.223,Z 208.824,A -85,B 0,C 180,E1 -27682.022,E2 -27682.022} C_VEL
LIN {X 0,Y 127.134,Z 202.583,A -85,B 0,C 180,E1 -27685.437,E2 -27685.437} C_VEL
LIN {X 0,Y 124.379,Z 197.49,A -85,B 0,C 180,E1 -27688.969,E2 -27688.969} C_VEL
LIN {X 0,Y 122.757,Z 194.742,A -85,B 0,C 180,E1 -27691.344,E2 -27691.344} C_VEL
LIN {X 0,Y 120.948,Z 191.628,A -85,B 0,C 180,E1 -27694.452,E2 -27694.452} C_VEL
LIN {X 0,Y 118.683,Z 187.765,A -85,B 0,C 180,E1 -27699.539,E2 -27699.539} C_VEL
LIN {X 0,Y 116.709,Z 184.243,A -85,B 0,C 180,E1 -27708.245,E2 -27708.245} C_VEL
LIN {X 0,Y 116.665,Z 183.052,A -85,B 0,C 180,E1 -27710.574,E2 -27710.574} C_VEL
LIN {X 0,Y 116.871,Z 183.159,A -85,B 0,C 180,E1 -27715.595,E2 -27715.595} C_VEL
LIN {X 0,Y 117.781,Z 186.346,A -85,B 0,C 180,E1 -27721.3,E2 -27721.3} C_VEL
LIN {X 0,Y 119.047,Z 187.972,A -85,B 0,C 180,E1 -27724.942,E2 -27724.942} C_VEL
LIN {X 0,Y 121.242,Z 191.77,A -85,B 0,C 180,E1 -27729.646,E2 -27729.646} C_VEL
LIN {X 0,Y 123.736,Z 196.282,A -85,B 0,C 180,E1 -27733.731,E2 -27733.731} C_VEL
LIN {X 0,Y 126.874,Z 202,A -85,B 0,C 180,E1 -27737.879,E2 -27737.879} C_VEL
LIN {X 0,Y 130.325,Z 209.176,A -85,B 0,C 180,E1 -27741.733,E2 -27741.733} C_VEL
LIN {X 0,Y 131.99,Z 213.091,A -85,B 0,C 180,E1 -27743.418,E2 -27743.418} C_VEL
LIN {X 0,Y 134.147,Z 220.675,A -85,B 0,C 180,E1 -27745.674,E2 -27745.674} C_VEL
LIN {X 0,Y 129.53,Z 268.685,A -85,B 0,C 180,E1 -27747.526,E2 -27747.526} C_VEL
LIN {X 0,Y 127.064,Z 282.637,A -85,B 0,C 180,E1 -27748.393,E2 -27748.393} C_VEL
LIN {X 0,Y 123.709,Z 295.689,A -85,B 0,C 180,E1 -27749.562,E2 -27749.562} C_VEL
LIN {X 0,Y 119.281,Z 309.133,A -85,B 0,C 180,E1 -27751.323,E2 -27751.323} C_VEL
LIN {X 0,Y 114.255,Z 321.323,A -85,B 0,C 180,E1 -27753.473,E2 -27753.473} C_VEL
LIN {X 0,Y 108.935,Z 332.638,A -85,B 0,C 180,E1 -27756.259,E2 -27756.259} C_VEL
LIN {X 0,Y 104.573,Z 340.518,A -85,B 0,C 180,E1 -27758.632,E2 -27758.632} C_VEL
LIN {X 0,Y 98.312,Z 351.049,A -85,B 0,C 180,E1 -27762.892,E2 -27762.892} C_VEL
LIN {X 0,Y 92.178,Z 360.525,A -85,B 0,C 180,E1 -27768.162,E2 -27768.162} C_VEL
LIN {X 0,Y 87.201,Z 367.936,A -85,B 0,C 180,E1 -27773.725,E2 -27773.725} C_VEL
LIN {X 0,Y 83.309,Z 373.873,A -85,B 0,C 180,E1 -27779.599,E2 -27779.599} C_VEL
LIN {X 0,Y 79.988,Z 379.434,A -85,B 0,C 180,E1 -27786.718,E2 -27786.718} C_VEL
LIN {X 0,Y 77.381,Z 385.237,A -85,B 0,C 180,E1 -27796.884,E2 -27796.884} C_VEL
LIN {X 0,Y 76.74,Z 388.512,A -85,B 0,C 180,E1 -27804.753,E2 -27804.753} C_VEL
LIN {X 0,Y 76.797,Z 390.199,A -85,B 0,C 180,E1 -27810.007,E2 -27810.007} C_VEL
LIN {X 0,Y 76.786,Z 391.5,A -85,B 0,C 180,E1 -27815.259,E2 -27815.259} C_VEL
LIN {X 0,Y 77.973,Z 393.082,A -85,B 0,C 180,E1 -27825.696,E2 -27825.696} C_VEL
LIN {X 0,Y 81.321,Z 393.368,A -85,B 0,C 180,E1 -27835.609,E2 -27835.609} C_VEL
LIN {X 0,Y 86.952,Z 392.384,A -85,B 0,C 180,E1 -27844.465,E2 -27844.465} C_VEL
LIN {X 0,Y 94.341,Z 390.109,A -85,B 0,C 180,E1 -27852.11,E2 -27852.11} C_VEL
LIN {X 0,Y 103.166,Z 386.486,A -85,B 0,C 180,E1 -27858.543,E2 -27858.543} C_VEL
LIN {X 0,Y 113.158,Z 381.411,A -85,B 0,C 180,E1 -27863.851,E2 -27863.851} C_VEL
LIN {X 0,Y 121.26,Z 376.538,A -85,B 0,C 180,E1 -27867.19,E2 -27867.19} C_VEL
LIN {X 0,Y 131.242,Z 369.563,A -85,B 0,C 180,E1 -27870.489,E2 -27870.489} C_VEL
LIN {X 0,Y 139.842,Z 362.47,A -85,B 0,C 180,E1 -27872.967,E2 -27872.967} C_VEL
LIN {X 0,Y 149.07,Z 353.65,A -85,B 0,C 180,E1 -27875.178,E2 -27875.178} C_VEL
LIN {X 0,Y 158.38,Z 343.184,A -85,B 0,C 180,E1 -27877.047,E2 -27877.047} C_VEL
LIN {X 0,Y 167.055,Z 331.514,A -85,B 0,C 180,E1 -27878.568,E2 -27878.568} C_VEL
LIN {X 0,Y 174.284,Z 319.828,A -85,B 0,C 180,E1 -27879.654,E2 -27879.654} C_VEL
LIN {X 0,Y 179.386,Z 309.884,A -85,B 0,C 180,E1 -27880.393,E2 -27880.393} C_VEL
LIN {X 0,Y 181.613,Z 304.686,A -85,B 0,C 180,E1 -27880.889,E2 -27880.889} C_VEL
LIN {X 0,Y 184.494,Z 296.069,A -85,B 0,C 180,E1 -27882.14,E2 -27882.14} C_VEL
LIN {X 0,Y 186.969,Z 287.294,A -85,B 0,C 180,E1 -27883.329,E2 -27883.329} C_VEL
LIN {X 0,Y 188.4,Z 281.745,A -85,B 0,C 180,E1 -27883.748,E2 -27883.748} C_VEL
LIN {X 0,Y 190.863,Z 270.632,A -85,B 0,C 180,E1 -27884.115,E2 -27884.115} C_VEL
LIN {X 0,Y 190.519,Z 268.486,A -85,B 0,C 180,E1 -27885.848,E2 -27885.848} C_VEL
LIN {X 0,Y 190.265,Z 267.373,A -85,B 0,C 180,E1 -27887.189,E2 -27887.189} C_VEL
LIN {X 0,Y 189.872,Z 264.822,A -85,B 0,C 180,E1 -27892.55,E2 -27892.55} C_VEL
LIN {X 0,Y 189.94,Z 265.129,A -85,B 0,C 180,E1 -27894.061,E2 -27894.061} C_VEL
LIN {X 0,Y 190.453,Z 267.758,A -85,B 0,C 180,E1 -27898.239,E2 -27898.239} C_VEL
LIN {X 0,Y 190.923,Z 269.771,A -85,B 0,C 180,E1 -27900.302,E2 -27900.302} C_VEL
LIN {X 0,Y 187.437,Z 284.265,A -85,B 0,C 180,E1 -27900.753,E2 -27900.753} C_VEL
LIN {X 0,Y 183.248,Z 296.624,A -85,B 0,C 180,E1 -27901.274,E2 -27901.274} C_VEL
LIN {X 0,Y 177.409,Z 310.032,A -85,B 0,C 180,E1 -27902.108,E2 -27902.108} C_VEL
LIN {X 0,Y 170.69,Z 322.237,A -85,B 0,C 180,E1 -27903.117,E2 -27903.117} C_VEL
LIN {X 0,Y 163.003,Z 333.671,A -85,B 0,C 180,E1 -27904.358,E2 -27904.358} C_VEL
LIN {X 0,Y 155.389,Z 343.204,A -85,B 0,C 180,E1 -27905.683,E2 -27905.683} C_VEL
LIN {X 0,Y 145.395,Z 353.704,A -85,B 0,C 180,E1 -27907.703,E2 -27907.703} C_VEL
LIN {X 0,Y 135.618,Z 362.337,A -85,B 0,C 180,E1 -27910.039,E2 -27910.039} C_VEL
LIN {X 0,Y 125.258,Z 370.011,A -85,B 0,C 180,E1 -27912.958,E2 -27912.958} C_VEL
LIN {X 0,Y 113.896,Z 376.991,A -85,B 0,C 180,E1 -27916.958,E2 -27916.958} C_VEL
LIN {X 0,Y 105.271,Z 381.373,A -85,B 0,C 180,E1 -27920.814,E2 -27920.814} C_VEL
LIN {X 0,Y 94.606,Z 385.711,A -85,B 0,C 180,E1 -27926.932,E2 -27926.932} C_VEL
LIN {X 0,Y 85.313,Z 388.472,A -85,B 0,C 180,E1 -27934.523,E2 -27934.523} C_VEL
LIN {X 0,Y 77.783,Z 389.709,A -85,B 0,C 180,E1 -27943.701,E2 -27943.701} C_VEL
LIN {X 0,Y 72.446,Z 389.482,A -85,B 0,C 180,E1 -27954.395,E2 -27954.395} C_VEL
LIN {X 0,Y 69.686,Z 387.82,A -85,B 0,C 180,E1 -27966.2,E2 -27966.2} C_VEL
LIN {X 0,Y 69.124,Z 386.46,A -85,B 0,C 180,E1 -27972.232,E2 -27972.232} C_VEL
LIN {X 0,Y 69.855,Z 382.642,A -85,B 0,C 180,E1 -27984.218,E2 -27984.218} C_VEL
LIN {X 0,Y 71.783,Z 378.76,A -85,B 0,C 180,E1 -27992.798,E2 -27992.798} C_VEL
LIN {X 0,Y 74.717,Z 373.983,A -85,B 0,C 180,E1 -28000.835,E2 -28000.835} C_VEL
LIN {X 0,Y 79.696,Z 367.038,A -85,B 0,C 180,E1 -28009.303,E2 -28009.303} C_VEL
LIN {X 0,Y 86.028,Z 358.424,A -85,B 0,C 180,E1 -28016.692,E2 -28016.692} C_VEL
LIN {X 0,Y 92.279,Z 349.441,A -85,B 0,C 180,E1 -28022.209,E2 -28022.209} C_VEL
LIN {X 0,Y 97.763,Z 340.584,A -85,B 0,C 180,E1 -28026.368,E2 -28026.368} C_VEL
LIN {X 0,Y 104.099,Z 329.9,A -85,B 0,C 180,E1 -28029.887,E2 -28029.887} C_VEL
LIN {X 0,Y 109.886,Z 318.309,A -85,B 0,C 180,E1 -28032.801,E2 -28032.801} C_VEL
LIN {X 0,Y 115.281,Z 305.561,A -85,B 0,C 180,E1 -28035.122,E2 -28035.122} C_VEL
LIN {X 0,Y 119.685,Z 292.43,A -85,B 0,C 180,E1 -28036.907,E2 -28036.907} C_VEL
LIN {X 0,Y 122.914,Z 279.759,A -85,B 0,C 180,E1 -28038.172,E2 -28038.172} C_VEL
LIN {X 0,Y 125.388,Z 266.603,A -85,B 0,C 180,E1 -28039.021,E2 -28039.021} C_VEL
LIN {X 0,Y 127.691,Z 246.672,A -85,B 0,C 180,E1 -28039.753,E2 -28039.753} C_VEL
LIN {X 0,Y 130.194,Z 221.045,A -85,B 0,C 180,E1 -28040.682,E2 -28040.682} C_VEL
LIN {X 0,Y 126.998,Z 213.175,A -85,B 0,C 180,E1 -28044.206,E2 -28044.206} C_VEL
LIN {X 0,Y 124.257,Z 207.263,A -85,B 0,C 180,E1 -28047.652,E2 -28047.652} C_VEL
LIN {X 0,Y 121.373,Z 201.683,A -85,B 0,C 180,E1 -28051.942,E2 -28051.942} C_VEL
LIN {X 0,Y 119.443,Z 198.264,A -85,B 0,C 180,E1 -28055.465,E2 -28055.465} C_VEL
LIN {X 0,Y 117.504,Z 194.625,A -85,B 0,C 180,E1 -28060.238,E2 -28060.238} C_VEL
LIN {X 0,Y 115.772,Z 191.166,A -85,B 0,C 180,E1 -28068.834,E2 -28068.834} C_VEL
LIN {X 0,Y 115.765,Z 190.022,A -85,B 0,C 180,E1 -28071.479,E2 -28071.479} C_VEL
LIN {X 0,Y 115.921,Z 190.215,A -85,B 0,C 180,E1 -28075.07,E2 -28075.07} C_VEL
LIN {X 0,Y 116.756,Z 193.315,A -85,B 0,C 180,E1 -28080.878,E2 -28080.878} C_VEL
LIN {X 0,Y 117.776,Z 194.793,A -85,B 0,C 180,E1 -28084.083,E2 -28084.083} C_VEL
LIN {X 0,Y 120.107,Z 199.212,A -85,B 0,C 180,E1 -28089.414,E2 -28089.414} C_VEL
LIN {X 0,Y 122.143,Z 203.153,A -85,B 0,C 180,E1 -28092.92,E2 -28092.92} C_VEL
LIN {X 0,Y 125.062,Z 208.984,A -85,B 0,C 180,E1 -28097.054,E2 -28097.054} C_VEL
LIN {X 0,Y 127.956,Z 215.529,A -85,B 0,C 180,E1 -28100.546,E2 -28100.546} C_VEL
LIN {X 0,Y 129.098,Z 218.808,A -85,B 0,C 180,E1 -28101.858,E2 -28101.858} C_VEL
LIN {X 0,Y 130.168,Z 222.97,A -85,B 0,C 180,E1 -28103.139,E2 -28103.139} C_VEL
LIN {X 0,Y 125.559,Z 268.85,A -85,B 0,C 180,E1 -28104.888,E2 -28104.888} C_VEL
LIN {X 0,Y 122.897,Z 283.135,A -85,B 0,C 180,E1 -28105.763,E2 -28105.763} C_VEL
LIN {X 0,Y 119.25,Z 296.583,A -85,B 0,C 180,E1 -28106.963,E2 -28106.963} C_VEL
LIN {X 0,Y 114.318,Z 310.694,A -85,B 0,C 180,E1 -28108.841,E2 -28108.841} C_VEL
LIN {X 0,Y 108.591,Z 323.63,A -85,B 0,C 180,E1 -28111.195,E2 -28111.195} C_VEL
LIN {X 0,Y 103.497,Z 333.593,A -85,B 0,C 180,E1 -28113.722,E2 -28113.722} C_VEL
LIN {X 0,Y 98.999,Z 341.358,A -85,B 0,C 180,E1 -28116.156,E2 -28116.156} C_VEL
LIN {X 0,Y 92.401,Z 351.675,A -85,B 0,C 180,E1 -28120.493,E2 -28120.493} C_VEL
LIN {X 0,Y 85.936,Z 361.005,A -85,B 0,C 180,E1 -28125.971,E2 -28125.971} C_VEL
LIN {X 0,Y 80.302,Z 368.747,A -85,B 0,C 180,E1 -28132.229,E2 -28132.229} C_VEL
LIN {X 0,Y 75.84,Z 375.197,A -85,B 0,C 180,E1 -28139.367,E2 -28139.367} C_VEL
LIN {X 0,Y 72.441,Z 380.455,A -85,B 0,C 180,E1 -28147.175,E2 -28147.175} C_VEL
LIN {X 0,Y 70.461,Z 384.721,A -85,B 0,C 180,E1 -28155.569,E2 -28155.569} C_VEL
LIN {X 0,Y 69.655,Z 388.086,A -85,B 0,C 180,E1 -28164.217,E2 -28164.217} C_VEL
LIN {X 0,Y 69.718,Z 389.818,A -85,B 0,C 180,E1 -28170.008,E2 -28170.008} C_VEL
LIN {X 0,Y 69.727,Z 391.161,A -85,B 0,C 180,E1 -28175.793,E2 -28175.793} C_VEL
LIN {X 0,Y 71.141,Z 392.823,A -85,B 0,C 180,E1 -28187.248,E2 -28187.248} C_VEL
LIN {X 0,Y 74.958,Z 393.192,A -85,B 0,C 180,E1 -28197.965,E2 -28197.965} C_VEL
LIN {X 0,Y 81.171,Z 392.29,A -85,B 0,C 180,E1 -28207.315,E2 -28207.315} C_VEL
LIN {X 0,Y 89.18,Z 390.099,A -85,B 0,C 180,E1 -28215.184,E2 -28215.184} C_VEL
LIN {X 0,Y 98.599,Z 386.563,A -85,B 0,C 180,E1 -28221.643,E2 -28221.643} C_VEL
LIN {X 0,Y 109.107,Z 381.58,A -85,B 0,C 180,E1 -28226.873,E2 -28226.873} C_VEL
LIN {X 0,Y 120.466,Z 375.001,A -85,B 0,C 180,E1 -28231.066,E2 -28231.066} C_VEL
LIN {X 0,Y 130.914,Z 367.729,A -85,B 0,C 180,E1 -28234.063,E2 -28234.063} C_VEL
LIN {X 0,Y 139.845,Z 360.299,A -85,B 0,C 180,E1 -28236.342,E2 -28236.342} C_VEL
LIN {X 0,Y 149.419,Z 351.104,A -85,B 0,C 180,E1 -28238.281,E2 -28238.281} C_VEL
LIN {X 0,Y 158.991,Z 340.169,A -85,B 0,C 180,E1 -28239.948,E2 -28239.948} C_VEL
LIN {X 0,Y 167.049,Z 329.079,A -85,B 0,C 180,E1 -28241.202,E2 -28241.202} C_VEL
LIN {X 0,Y 174.431,Z 316.837,A -85,B 0,C 180,E1 -28242.162,E2 -28242.162} C_VEL
LIN {X 0,Y 180.188,Z 305.128,A -85,B 0,C 180,E1 -28242.87,E2 -28242.87} C_VEL
LIN {X 0,Y 185.403,Z 291.649,A -85,B 0,C 180,E1 -28243.46,E2 -28243.46} C_VEL
LIN {X 0,Y 188.4,Z 281.745,A -85,B 0,C 180,E1 -28243.748,E2 -28243.748} C_VEL
LIN {X 0,Y 188.931,Z 279.278,A -85,B 0,C 180,E1 -28244.092,E2 -28244.092} C_VEL
LIN {X 0,Y 189.162,Z 277.002,A -85,B 0,C 180,E1 -28244.905,E2 -28244.905} C_VEL
LIN {X 0,Y 189.091,Z 275.422,A -85,B 0,C 180,E1 -28246.014,E2 -28246.014} C_VEL
LIN {X 0,Y 188.52,Z 273.21,A -85,B 0,C 180,E1 -28249.683,E2 -28249.683} C_VEL
LIN {X 0,Y 188.561,Z 271.849,A -85,B 0,C 180,E1 -28252.498,E2 -28252.498} C_VEL
LIN {X 0,Y 188.602,Z 272.217,A -85,B 0,C 180,E1 -28254.111,E2 -28254.111} C_VEL
LIN {X 0,Y 188.858,Z 274.496,A -85,B 0,C 180,E1 -28257.738,E2 -28257.738} C_VEL
LIN {X 0,Y 188.917,Z 275.054,A -85,B 0,C 180,E1 -28258.313,E2 -28258.313} C_VEL
LIN {X 0,Y 185.011,Z 289.012,A -85,B 0,C 180,E1 -28258.751,E2 -28258.751} C_VEL
LIN {X 0,Y 180.113,Z 301.913,A -85,B 0,C 180,E1 -28259.335,E2 -28259.335} C_VEL
LIN {X 0,Y 173.944,Z 314.633,A -85,B 0,C 180,E1 -28260.136,E2 -28260.136} C_VEL
LIN {X 0,Y 166.083,Z 327.604,A -85,B 0,C 180,E1 -28261.222,E2 -28261.222} C_VEL
LIN {X 0,Y 157.198,Z 339.434,A -85,B 0,C 180,E1 -28262.554,E2 -28262.554} C_VEL
LIN {X 0,Y 147.982,Z 349.633,A -85,B 0,C 180,E1 -28264.137,E2 -28264.137} C_VEL
LIN {X 0,Y 138.765,Z 358.243,A -85,B 0,C 180,E1 -28265.945,E2 -28265.945} C_VEL
LIN {X 0,Y 127.901,Z 366.748,A -85,B 0,C 180,E1 -28268.449,E2 -28268.449} C_VEL
LIN {X 0,Y 118.214,Z 373.12,A -85,B 0,C 180,E1 -28271.178,E2 -28271.178} C_VEL
LIN {X 0,Y 106.537,Z 379.445,A -85,B 0,C 180,E1 -28275.286,E2 -28275.286} C_VEL
LIN {X 0,Y 97.001,Z 383.611,A -85,B 0,C 180,E1 -28279.613,E2 -28279.613} C_VEL
LIN {X 0,Y 86.148,Z 387.253,A -85,B 0,C 180,E1 -28286.17,E2 -28286.17} C_VEL
LIN {X 0,Y 76.751,Z 389.368,A -85,B 0,C 180,E1 -28294.488,E2 -28294.488} C_VEL
LIN {X 0,Y 69.29,Z 390.006,A -85,B 0,C 180,E1 -28304.753,E2 -28304.753} C_VEL
LIN {X 0,Y 64.312,Z 389.167,A -85,B 0,C 180,E1 -28316.869,E2 -28316.869} C_VEL
LIN {X 0,Y 62.922,Z 388.206,A -85,B 0,C 180,E1 -28323.453,E2 -28323.453} C_VEL
LIN {X 0,Y 62.133,Z 386.893,A -85,B 0,C 180,E1 -28330.154,E2 -28330.154} C_VEL
LIN {X 0,Y 62.576,Z 383.179,A -85,B 0,C 180,E1 -28343.542,E2 -28343.542} C_VEL
LIN {X 0,Y 64.59,Z 379.4,A -85,B 0,C 180,E1 -28353.11,E2 -28353.11} C_VEL
LIN {X 0,Y 67.7,Z 374.722,A -85,B 0,C 180,E1 -28361.974,E2 -28361.974} C_VEL
LIN {X 0,Y 72.955,Z 367.925,A -85,B 0,C 180,E1 -28371.168,E2 -28371.168} C_VEL
LIN {X 0,Y 78.68,Z 360.797,A -85,B 0,C 180,E1 -28377.958,E2 -28377.958} C_VEL
LIN {X 0,Y 85.213,Z 352.13,A -85,B 0,C 180,E1 -28383.945,E2 -28383.945} C_VEL
LIN {X 0,Y 92.134,Z 341.973,A -85,B 0,C 180,E1 -28388.991,E2 -28388.991} C_VEL
LIN {X 0,Y 98.681,Z 331.552,A -85,B 0,C 180,E1 -28392.569,E2 -28392.569} C_VEL
LIN {X 0,Y 104.788,Z 320.246,A -85,B 0,C 180,E1 -28395.439,E2 -28395.439} C_VEL
LIN {X 0,Y 110.389,Z 307.908,A -85,B 0,C 180,E1 -28397.733,E2 -28397.733} C_VEL
LIN {X 0,Y 114.971,Z 295.365,A -85,B 0,C 180,E1 -28399.481,E2 -28399.481} C_VEL
LIN {X 0,Y 118.936,Z 281.076,A -85,B 0,C 180,E1 -28400.924,E2 -28400.924} C_VEL
LIN {X 0,Y 121.666,Z 267.361,A -85,B 0,C 180,E1 -28401.807,E2 -28401.807} C_VEL
LIN {X 0,Y 124.022,Z 248.041,A -85,B 0,C 180,E1 -28402.491,E2 -28402.491} C_VEL
LIN {X 0,Y 126.455,Z 223.976,A -85,B 0,C 180,E1 -28403.344,E2 -28403.344} C_VEL
LIN {X 0,Y 123.422,Z 216.15,A -85,B 0,C 180,E1 -28407.25,E2 -28407.25} C_VEL
LIN {X 0,Y 120.487,Z 209.849,A -85,B 0,C 180,E1 -28411.674,E2 -28411.674} C_VEL
LIN {X 0,Y 118.091,Z 205.031,A -85,B 0,C 180,E1 -28416.268,E2 -28416.268} C_VEL
LIN {X 0,Y 116.159,Z 201.292,A -85,B 0,C 180,E1 -28421.515,E2 -28421.515} C_VEL
LIN {X 0,Y 114.844,Z 197.585,A -85,B 0,C 180,E1 -28430.547,E2 -28430.547} C_VEL
LIN {X 0,Y 114.875,Z 197.126,A -85,B 0,C 180,E1 -28431.413,E2 -28431.413} C_VEL
LIN {X 0,Y 114.988,Z 197.394,A -85,B 0,C 180,E1 -28434.784,E2 -28434.784} C_VEL
LIN {X 0,Y 115.847,Z 200.474,A -85,B 0,C 180,E1 -28440.885,E2 -28440.885} C_VEL
LIN {X 0,Y 116.484,Z 201.47,A -85,B 0,C 180,E1 -28443.04,E2 -28443.04} C_VEL
LIN {X 0,Y 118.555,Z 205.785,A -85,B 0,C 180,E1 -28448.319,E2 -28448.319} C_VEL
LIN {X 0,Y 120.435,Z 209.735,A -85,B 0,C 180,E1 -28451.856,E2 -28451.856} C_VEL
LIN {X 0,Y 123.282,Z 215.915,A -85,B 0,C 180,E1 -28456.202,E2 -28456.202} C_VEL
LIN {X 0,Y 125.702,Z 222.128,A -85,B 0,C 180,E1 -28459.399,E2 -28459.399} C_VEL
LIN {X 0,Y 126.478,Z 225.47,A -85,B 0,C 180,E1 -28460.491,E2 -28460.491} C_VEL
LIN {X 0,Y 121.879,Z 269.013,A -85,B 0,C 180,E1 -28462.09,E2 -28462.09} C_VEL
LIN {X 0,Y 119.011,Z 283.64,A -85,B 0,C 180,E1 -28462.961,E2 -28462.961} C_VEL
LIN {X 0,Y 115.062,Z 297.483,A -85,B 0,C 180,E1 -28464.177,E2 -28464.177} C_VEL
LIN {X 0,Y 110.302,Z 310.456,A -85,B 0,C 180,E1 -28465.857,E2 -28465.857} C_VEL
LIN {X 0,Y 104.272,Z 323.542,A -85,B 0,C 180,E1 -28468.165,E2 -28468.165} C_VEL
LIN {X 0,Y 98.995,Z 333.392,A -85,B 0,C 180,E1 -28470.623,E2 -28470.623} C_VEL
LIN {X 0,Y 94.275,Z 341.139,A -85,B 0,C 180,E1 -28473.013,E2 -28473.013} C_VEL
LIN {X 0,Y 86.697,Z 352.293,A -85,B 0,C 180,E1 -28477.791,E2 -28477.791} C_VEL
LIN {X 0,Y 79.841,Z 361.485,A -85,B 0,C 180,E1 -28483.442,E2 -28483.442} C_VEL
LIN {X 0,Y 74.124,Z 368.729,A -85,B 0,C 180,E1 -28489.63,E2 -28489.63} C_VEL
LIN {X 0,Y 69.734,Z 374.484,A -85,B 0,C 180,E1 -28496.347,E2 -28496.347} C_VEL
LIN {X 0,Y 65.9,Z 379.84,A -85,B 0,C 180,E1 -28504.759,E2 -28504.759} C_VEL
LIN {X 0,Y 63.105,Z 385.461,A -85,B 0,C 180,E1 -28517.139,E2 -28517.139} C_VEL
LIN {X 0,Y 62.584,Z 387.645,A -85,B 0,C 180,E1 -28523.562,E2 -28523.562} C_VEL
LIN {X 0,Y 62.628,Z 389.433,A -85,B 0,C 180,E1 -28530.009,E2 -28530.009} C_VEL
LIN {X 0,Y 62.649,Z 390.82,A -85,B 0,C 180,E1 -28536.45,E2 -28536.45} C_VEL
LIN {X 0,Y 64.377,Z 392.565,A -85,B 0,C 180,E1 -28549.127,E2 -28549.127} C_VEL
LIN {X 0,Y 68.749,Z 393.016,A -85,B 0,C 180,E1 -28560.749,E2 -28560.749} C_VEL
LIN {X 0,Y 75.623,Z 392.196,A -85,B 0,C 180,E1 -28570.592,E2 -28570.592} C_VEL
LIN {X 0,Y 84.296,Z 390.088,A -85,B 0,C 180,E1 -28578.631,E2 -28578.631} C_VEL
LIN {X 0,Y 94.336,Z 386.641,A -85,B 0,C 180,E1 -28585.044,E2 -28585.044} C_VEL
LIN {X 0,Y 105.385,Z 381.762,A -85,B 0,C 180,E1 -28590.117,E2 -28590.117} C_VEL
LIN {X 0,Y 117.202,Z 375.297,A -85,B 0,C 180,E1 -28594.099,E2 -28594.099} C_VEL
LIN {X 0,Y 127.969,Z 368.141,A -85,B 0,C 180,E1 -28596.922,E2 -28596.922} C_VEL
LIN {X 0,Y 137.326,Z 360.704,A -85,B 0,C 180,E1 -28599.076,E2 -28599.076} C_VEL
LIN {X 0,Y 146.952,Z 351.792,A -85,B 0,C 180,E1 -28600.841,E2 -28600.841} C_VEL
LIN {X 0,Y 155.075,Z 342.972,A -85,B 0,C 180,E1 -28602.134,E2 -28602.134} C_VEL
LIN {X 0,Y 164.1,Z 331.337,A -85,B 0,C 180,E1 -28603.399,E2 -28603.399} C_VEL
LIN {X 0,Y 171.572,Z 319.698,A -85,B 0,C 180,E1 -28604.295,E2 -28604.295} C_VEL
LIN {X 0,Y 177.4,Z 308.668,A -85,B 0,C 180,E1 -28604.951,E2 -28604.951} C_VEL
LIN {X 0,Y 183.256,Z 294.821,A -85,B 0,C 180,E1 -28605.527,E2 -28605.527} C_VEL
LIN {X 0,Y 187.763,Z 280.534,A -85,B 0,C 180,E1 -28605.93,E2 -28605.93} C_VEL
LIN {X 0,Y 188.953,Z 275.412,A -85,B 0,C 180,E1 -28606.143,E2 -28606.143} C_VEL
LIN {X 0,Y 188.716,Z 274.041,A -85,B 0,C 180,E1 -28607.901,E2 -28607.901} C_VEL
LIN {X 0,Y 188.52,Z 273.21,A -85,B 0,C 180,E1 -28609.683,E2 -28609.683} C_VEL
LIN {X 0,Y 188.34,Z 273.304,A -85,B 0,C 180,E1 -28610.863,E2 -28610.863} C_VEL
LIN {X 0,Y 187.968,Z 274.549,A -85,B 0,C 180,E1 -28612.005,E2 -28612.005} C_VEL
LIN {X 0,Y 186.979,Z 279.453,A -85,B 0,C 180,E1 -28614.997,E2 -28614.997} C_VEL
LIN {X 0,Y 186.912,Z 280.195,A -85,B 0,C 180,E1 -28615.808,E2 -28615.808} C_VEL
LIN {X 0,Y 186.938,Z 280.464,A -85,B 0,C 180,E1 -28616.288,E2 -28616.288} C_VEL
LIN {X 0,Y 182.468,Z 294.327,A -85,B 0,C 180,E1 -28616.729,E2 -28616.729} C_VEL
LIN {X 0,Y 176.773,Z 307.633,A -85,B 0,C 180,E1 -28617.374,E2 -28617.374} C_VEL
LIN {X 0,Y 170.084,Z 319.968,A -85,B 0,C 180,E1 -28618.165,E2 -28618.165} C_VEL
LIN {X 0,Y 162.551,Z 331.296,A -85,B 0,C 180,E1 -28619.102,E2 -28619.102} C_VEL
LIN {X 0,Y 153.748,Z 342.266,A -85,B 0,C 180,E1 -28620.296,E2 -28620.296} C_VEL
LIN {X 0,Y 144.153,Z 352.229,A -85,B 0,C 180,E1 -28621.78,E2 -28621.78} C_VEL
LIN {X 0,Y 133.819,Z 361.215,A -85,B 0,C 180,E1 -28623.695,E2 -28623.695} C_VEL
LIN {X 0,Y 123.648,Z 368.592,A -85,B 0,C 180,E1 -28625.874,E2 -28625.874} C_VEL
LIN {X 0,Y 113.696,Z 374.648,A -85,B 0,C 180,E1 -28628.465,E2 -28628.465} C_VEL
LIN {X 0,Y 103.566,Z 379.787,A -85,B 0,C 180,E1 -28631.733,E2 -28631.733} C_VEL
LIN {X 0,Y 91.725,Z 384.587,A -85,B 0,C 180,E1 -28636.692,E2 -28636.692} C_VEL
LIN {X 0,Y 83.088,Z 387.235,A -85,B 0,C 180,E1 -28641.48,E2 -28641.48} C_VEL
LIN {X 0,Y 72.729,Z 389.448,A -85,B 0,C 180,E1 -28649.562,E2 -28649.562} C_VEL
LIN {X 0,Y 64.195,Z 390.199,A -85,B 0,C 180,E1 -28659.959,E2 -28659.959} C_VEL
LIN {X 0,Y 58.16,Z 389.499,A -85,B 0,C 180,E1 -28672.817,E2 -28672.817} C_VEL
LIN {X 0,Y 56.1,Z 388.402,A -85,B 0,C 180,E1 -28681.221,E2 -28681.221} C_VEL
LIN {X 0,Y 54.844,Z 385.708,A -85,B 0,C 180,E1 -28695.139,E2 -28695.139} C_VEL
LIN {X 0,Y 56.221,Z 381.918,A -85,B 0,C 180,E1 -28708.377,E2 -28708.377} C_VEL
LIN {X 0,Y 59.456,Z 377.06,A -85,B 0,C 180,E1 -28720.203,E2 -28720.203} C_VEL
LIN {X 0,Y 64.568,Z 370.804,A -85,B 0,C 180,E1 -28730.707,E2 -28730.707} C_VEL
LIN {X 0,Y 71.352,Z 362.999,A -85,B 0,C 180,E1 -28739.495,E2 -28739.495} C_VEL
LIN {X 0,Y 77.696,Z 355.421,A -85,B 0,C 180,E1 -28745.409,E2 -28745.409} C_VEL
LIN {X 0,Y 84.224,Z 346.875,A -85,B 0,C 180,E1 -28750.283,E2 -28750.283} C_VEL
LIN {X 0,Y 90.742,Z 337.445,A -85,B 0,C 180,E1 -28754.182,E2 -28754.182} C_VEL
LIN {X 0,Y 97.044,Z 327.285,A -85,B 0,C 180,E1 -28757.151,E2 -28757.151} C_VEL
LIN {X 0,Y 103.553,Z 314.955,A -85,B 0,C 180,E1 -28759.767,E2 -28759.767} C_VEL
LIN {X 0,Y 108.691,Z 303.132,A -85,B 0,C 180,E1 -28761.62,E2 -28761.62} C_VEL
LIN {X 0,Y 113.427,Z 289.064,A -85,B 0,C 180,E1 -28763.275,E2 -28763.275} C_VEL
LIN {X 0,Y 116.943,Z 275.09,A -85,B 0,C 180,E1 -28764.367,E2 -28764.367} C_VEL
LIN {X 0,Y 119.234,Z 261.652,A -85,B 0,C 180,E1 -28765.018,E2 -28765.018} C_VEL
LIN {X 0,Y 122.867,Z 228.548,A -85,B 0,C 180,E1 -28766.072,E2 -28766.072} C_VEL
LIN {X 0,Y 122.897,Z 226.83,A -85,B 0,C 180,E1 -28766.281,E2 -28766.281} C_VEL
LIN {X 0,Y 120.669,Z 220.859,A -85,B 0,C 180,E1 -28769.6,E2 -28769.6} C_VEL
LIN {X 0,Y 118.528,Z 215.802,A -85,B 0,C 180,E1 -28773.295,E2 -28773.295} C_VEL
LIN {X 0,Y 116.463,Z 211.317,A -85,B 0,C 180,E1 -28777.796,E2 -28777.796} C_VEL
LIN {X 0,Y 115.036,Z 208.17,A -85,B 0,C 180,E1 -28782.226,E2 -28782.226} C_VEL
LIN {X 0,Y 113.964,Z 204.393,A -85,B 0,C 180,E1 -28791.454,E2 -28791.454} C_VEL
LIN {X 0,Y 114.055,Z 204.198,A -85,B 0,C 180,E1 -28793.838,E2 -28793.838} C_VEL
LIN {X 0,Y 114.828,Z 207.45,A -85,B 0,C 180,E1 -28800.452,E2 -28800.452} C_VEL
LIN {X 0,Y 115.347,Z 208.5,A -85,B 0,C 180,E1 -28802.418,E2 -28802.418} C_VEL
LIN {X 0,Y 117.019,Z 212.281,A -85,B 0,C 180,E1 -28807.127,E2 -28807.127} C_VEL
LIN {X 0,Y 119.139,Z 217.071,A -85,B 0,C 180,E1 -28811.428,E2 -28811.428} C_VEL
LIN {X 0,Y 121.67,Z 223.45,A -85,B 0,C 180,E1 -28815.573,E2 -28815.573} C_VEL
LIN {X 0,Y 123.048,Z 227.646,A -85,B 0,C 180,E1 -28817.62,E2 -28817.62} C_VEL
LIN {X 0,Y 119.069,Z 265.028,A -85,B 0,C 180,E1 -28818.926,E2 -28818.926} C_VEL
LIN {X 0,Y 116.59,Z 279.294,A -85,B 0,C 180,E1 -28819.659,E2 -28819.659} C_VEL
LIN {X 0,Y 113.065,Z 292.462,A -85,B 0,C 180,E1 -28820.583,E2 -28820.583} C_VEL
LIN {X 0,Y 108.132,Z 306.641,A -85,B 0,C 180,E1 -28822.17,E2 -28822.17} C_VEL
LIN {X 0,Y 102.092,Z 319.921,A -85,B 0,C 180,E1 -28824.213,E2 -28824.213} C_VEL
LIN {X 0,Y 96.672,Z 330.143,A -85,B 0,C 180,E1 -28826.461,E2 -28826.461} C_VEL
LIN {X 0,Y 90.54,Z 339.851,A -85,B 0,C 180,E1 -28829.174,E2 -28829.174} C_VEL
LIN {X 0,Y 83.797,Z 349.5,A -85,B 0,C 180,E1 -28833.011,E2 -28833.011} C_VEL
LIN {X 0,Y 76.267,Z 359.164,A -85,B 0,C 180,E1 -28838.451,E2 -28838.451} C_VEL
LIN {X 0,Y 69.409,Z 367.323,A -85,B 0,C 180,E1 -28845.161,E2 -28845.161} C_VEL
LIN {X 0,Y 63.881,Z 373.764,A -85,B 0,C 180,E1 -28852.776,E2 -28852.776} C_VEL
LIN {X 0,Y 59.5,Z 379.226,A -85,B 0,C 180,E1 -28861.816,E2 -28861.816} C_VEL
LIN {X 0,Y 56.153,Z 384.943,A -85,B 0,C 180,E1 -28875.514,E2 -28875.514} C_VEL
LIN {X 0,Y 55.538,Z 387.178,A -85,B 0,C 180,E1 -28882.741,E2 -28882.741} C_VEL
LIN {X 0,Y 55.528,Z 389.019,A -85,B 0,C 180,E1 -28890.01,E2 -28890.01} C_VEL
LIN {X 0,Y 55.586,Z 390.458,A -85,B 0,C 180,E1 -28897.274,E2 -28897.274} C_VEL
LIN {X 0,Y 57.671,Z 392.296,A -85,B 0,C 180,E1 -28911.455,E2 -28911.455} C_VEL
LIN {X 0,Y 62.736,Z 392.835,A -85,B 0,C 180,E1 -28924.075,E2 -28924.075} C_VEL
LIN {X 0,Y 70.363,Z 392.1,A -85,B 0,C 180,E1 -28934.372,E2 -28934.372} C_VEL
LIN {X 0,Y 79.762,Z 390.085,A -85,B 0,C 180,E1 -28942.479,E2 -28942.479} C_VEL
LIN {X 0,Y 90.444,Z 386.736,A -85,B 0,C 180,E1 -28948.744,E2 -28948.744} C_VEL
LIN {X 0,Y 102.026,Z 381.955,A -85,B 0,C 180,E1 -28953.584,E2 -28953.584} C_VEL
LIN {X 0,Y 114.287,Z 375.594,A -85,B 0,C 180,E1 -28957.294,E2 -28957.294} C_VEL
LIN {X 0,Y 125.363,Z 368.553,A -85,B 0,C 180,E1 -28959.901,E2 -28959.901} C_VEL
LIN {X 0,Y 134.963,Z 361.244,A -85,B 0,C 180,E1 -28961.881,E2 -28961.881} C_VEL
LIN {X 0,Y 144.79,Z 352.48,A -85,B 0,C 180,E1 -28963.478,E2 -28963.478} C_VEL
LIN {X 0,Y 154.728,Z 341.9,A -85,B 0,C 180,E1 -28964.855,E2 -28964.855} C_VEL
LIN {X 0,Y 163.067,Z 331.251,A -85,B 0,C 180,E1 -28965.878,E2 -28965.878} C_VEL
LIN {X 0,Y 170.649,Z 319.633,A -85,B 0,C 180,E1 -28966.662,E2 -28966.662} C_VEL
LIN {X 0,Y 176.559,Z 308.628,A -85,B 0,C 180,E1 -28967.235,E2 -28967.235} C_VEL
LIN {X 0,Y 181.997,Z 296.096,A -85,B 0,C 180,E1 -28967.698,E2 -28967.698} C_VEL
LIN {X 0,Y 186.617,Z 282.083,A -85,B 0,C 180,E1 -28968.054,E2 -28968.054} C_VEL
LIN {X 0,Y 186.949,Z 280.851,A -85,B 0,C 180,E1 -28968.152,E2 -28968.152} C_VEL
LIN {X 0,Y 186.919,Z 278.816,A -85,B 0,C 180,E1 -28972.431,E2 -28972.431} C_VEL
LIN {X 0,Y 186.938,Z 279.038,A -85,B 0,C 180,E1 -28973.788,E2 -28973.788} C_VEL
LIN {X 0,Y 186.912,Z 280.195,A -85,B 0,C 180,E1 -28975.808,E2 -28975.808} C_VEL
LIN {X 0,Y 186.735,Z 281.065,A -85,B 0,C 180,E1 -28976.147,E2 -28976.147} C_VEL
LIN {X 0,Y 186.051,Z 283.54,A -85,B 0,C 180,E1 -28976.318,E2 -28976.318} C_VEL
LIN {X 0,Y 184.919,Z 287.036,A -85,B 0,C 180,E1 -28976.087,E2 -28976.087} C_VEL
LIN {X 0,Y 181.722,Z 295.438,A -85,B 0,C 180,E1 -28974.9,E2 -28974.9} C_VEL
LIN {X 0,Y 180.151,Z 299.221,A -85,B 0,C 180,E1 -28974.696,E2 -28974.696} C_VEL
LIN {X 0,Y 179.821,Z 299.97,A -85,B 0,C 180,E1 -28974.71,E2 -28974.71} C_VEL
LIN {X 0,Y 173.444,Z 313.213,A -85,B 0,C 180,E1 -28975.344,E2 -28975.344} C_VEL
LIN {X 0,Y 165.534,Z 326.232,A -85,B 0,C 180,E1 -28976.184,E2 -28976.184} C_VEL
LIN {X 0,Y 157.37,Z 337.19,A -85,B 0,C 180,E1 -28977.114,E2 -28977.114} C_VEL
LIN {X 0,Y 147.66,Z 348.001,A -85,B 0,C 180,E1 -28978.325,E2 -28978.325} C_VEL
LIN {X 0,Y 138.077,Z 356.892,A -85,B 0,C 180,E1 -28979.732,E2 -28979.732} C_VEL
LIN {X 0,Y 126.571,Z 365.797,A -85,B 0,C 180,E1 -28981.732,E2 -28981.732} C_VEL
LIN {X 0,Y 115.585,Z 372.784,A -85,B 0,C 180,E1 -28984.037,E2 -28984.037} C_VEL
LIN {X 0,Y 103.178,Z 379.162,A -85,B 0,C 180,E1 -28987.307,E2 -28987.307} C_VEL
LIN {X 0,Y 93.022,Z 383.37,A -85,B 0,C 180,E1 -28990.803,E2 -28990.803} C_VEL
LIN {X 0,Y 80.623,Z 387.219,A -85,B 0,C 180,E1 -28996.463,E2 -28996.463} C_VEL
LIN {X 0,Y 69.3,Z 389.533,A -85,B 0,C 180,E1 -29004.096,E2 -29004.096} C_VEL
LIN {X 0,Y 59.616,Z 390.382,A -85,B 0,C 180,E1 -29014.373,E2 -29014.373} C_VEL
LIN {X 0,Y 52.349,Z 389.792,A -85,B 0,C 180,E1 -29027.821,E2 -29027.821} C_VEL
LIN {X 0,Y 49.327,Z 388.55,A -85,B 0,C 180,E1 -29038.689,E2 -29038.689} C_VEL
LIN {X 0,Y 47.753,Z 386.194,A -85,B 0,C 180,E1 -29052.869,E2 -29052.869} C_VEL
LIN {X 0,Y 49.3,Z 381.928,A -85,B 0,C 180,E1 -29069.988,E2 -29069.988} C_VEL
LIN {X 0,Y 52.398,Z 377.755,A -85,B 0,C 180,E1 -29081.595,E2 -29081.595} C_VEL
LIN {X 0,Y 56.997,Z 372.57,A -85,B 0,C 180,E1 -29091.7,E2 -29091.7} C_VEL
LIN {X 0,Y 64.133,Z 365.162,A -85,B 0,C 180,E1 -29101.357,E2 -29101.357} C_VEL
LIN {X 0,Y 71.831,Z 356.755,A -85,B 0,C 180,E1 -29108.521,E2 -29108.521} C_VEL
LIN {X 0,Y 78.954,Z 348.122,A -85,B 0,C 180,E1 -29113.608,E2 -29113.608} C_VEL
LIN {X 0,Y 86.491,Z 337.868,A -85,B 0,C 180,E1 -29117.846,E2 -29117.846} C_VEL
LIN {X 0,Y 93.808,Z 326.504,A -85,B 0,C 180,E1 -29121.003,E2 -29121.003} C_VEL
LIN {X 0,Y 100.631,Z 313.903,A -85,B 0,C 180,E1 -29123.422,E2 -29123.422} C_VEL
LIN {X 0,Y 105.963,Z 301.768,A -85,B 0,C 180,E1 -29125.152,E2 -29125.152} C_VEL
LIN {X 0,Y 110.684,Z 287.902,A -85,B 0,C 180,E1 -29126.629,E2 -29126.629} C_VEL
LIN {X 0,Y 113.819,Z 275.596,A -85,B 0,C 180,E1 -29127.544,E2 -29127.544} C_VEL
LIN {X 0,Y 116.332,Z 261.353,A -85,B 0,C 180,E1 -29128.16,E2 -29128.16} C_VEL
LIN {X 0,Y 119.731,Z 231.251,A -85,B 0,C 180,E1 -29129.05,E2 -29129.05} C_VEL
LIN {X 0,Y 119.709,Z 229.988,A -85,B 0,C 180,E1 -29129.275,E2 -29129.275} C_VEL
LIN {X 0,Y 117.803,Z 224.604,A -85,B 0,C 180,E1 -29132.657,E2 -29132.657} C_VEL
LIN {X 0,Y 116.049,Z 220.287,A -85,B 0,C 180,E1 -29136.364,E2 -29136.364} C_VEL
LIN {X 0,Y 114.97,Z 217.741,A -85,B 0,C 180,E1 -29139.211,E2 -29139.211} C_VEL
LIN {X 0,Y 113.939,Z 215.077,A -85,B 0,C 180,E1 -29142.913,E2 -29142.913} C_VEL
LIN {X 0,Y 113.13,Z 211.166,A -85,B 0,C 180,E1 -29152.875,E2 -29152.875} C_VEL
LIN {X 0,Y 114.12,Z 215.188,A -85,B 0,C 180,E1 -29161.342,E2 -29161.342} C_VEL
LIN {X 0,Y 115.661,Z 219.088,A -85,B 0,C 180,E1 -29166.235,E2 -29166.235} C_VEL
LIN {X 0,Y 117.757,Z 224.546,A -85,B 0,C 180,E1 -29170.888,E2 -29170.888} C_VEL
LIN {X 0,Y 119.525,Z 229.483,A -85,B 0,C 180,E1 -29174.048,E2 -29174.048} C_VEL
LIN {X 0,Y 119.879,Z 230.552,A -85,B 0,C 180,E1 -29174.638,E2 -29174.638} C_VEL
LIN {X 0,Y 116.136,Z 264.621,A -85,B 0,C 180,E1 -29175.775,E2 -29175.775} C_VEL
LIN {X 0,Y 113.606,Z 278.853,A -85,B 0,C 180,E1 -29176.455,E2 -29176.455} C_VEL
LIN {X 0,Y 109.951,Z 292.205,A -85,B 0,C 180,E1 -29177.313,E2 -29177.313} C_VEL
LIN {X 0,Y 104.848,Z 306.404,A -85,B 0,C 180,E1 -29178.79,E2 -29178.79} C_VEL
LIN {X 0,Y 98.595,Z 319.695,A -85,B 0,C 180,E1 -29180.696,E2 -29180.696} C_VEL
LIN {X 0,Y 93.865,Z 328.245,A -85,B 0,C 180,E1 -29182.392,E2 -29182.392} C_VEL
LIN {X 0,Y 88.711,Z 336.357,A -85,B 0,C 180,E1 -29184.363,E2 -29184.363} C_VEL
LIN {X 0,Y 81.534,Z 346.57,A -85,B 0,C 180,E1 -29187.946,E2 -29187.946} C_VEL
LIN {X 0,Y 73.31,Z 356.679,A -85,B 0,C 180,E1 -29192.997,E2 -29192.997} C_VEL
LIN {X 0,Y 65.847,Z 365.059,A -85,B 0,C 180,E1 -29199.317,E2 -29199.317} C_VEL
LIN {X 0,Y 59.331,Z 372.021,A -85,B 0,C 180,E1 -29207.083,E2 -29207.083} C_VEL
LIN {X 0,Y 53.299,Z 378.612,A -85,B 0,C 180,E1 -29218.18,E2 -29218.18} C_VEL
LIN {X 0,Y 49.956,Z 383.165,A -85,B 0,C 180,E1 -29229.42,E2 -29229.42} C_VEL
LIN {X 0,Y 48.492,Z 386.709,A -85,B 0,C 180,E1 -29241.679,E2 -29241.679} C_VEL
LIN {X 0,Y 48.445,Z 388.596,A -85,B 0,C 180,E1 -29250.012,E2 -29250.012} C_VEL
LIN {X 0,Y 48.553,Z 390.076,A -85,B 0,C 180,E1 -29258.335,E2 -29258.335} C_VEL
LIN {X 0,Y 51.086,Z 391.999,A -85,B 0,C 180,E1 -29274.387,E2 -29274.387} C_VEL
LIN {X 0,Y 56.957,Z 392.623,A -85,B 0,C 180,E1 -29288.107,E2 -29288.107} C_VEL
LIN {X 0,Y 65.443,Z 391.98,A -85,B 0,C 180,E1 -29298.754,E2 -29298.754} C_VEL
LIN {X 0,Y 75.63,Z 390.064,A -85,B 0,C 180,E1 -29306.768,E2 -29306.768} C_VEL
LIN {X 0,Y 86.969,Z 386.824,A -85,B 0,C 180,E1 -29312.751,E2 -29312.751} C_VEL
LIN {X 0,Y 99.065,Z 382.148,A -85,B 0,C 180,E1 -29317.273,E2 -29317.273} C_VEL
LIN {X 0,Y 111.746,Z 375.89,A -85,B 0,C 180,E1 -29320.644,E2 -29320.644} C_VEL
LIN {X 0,Y 123.104,Z 368.967,A -85,B 0,C 180,E1 -29323.006,E2 -29323.006} C_VEL
LIN {X 0,Y 134.593,Z 360.441,A -85,B 0,C 180,E1 -29325.033,E2 -29325.033} C_VEL
LIN {X 0,Y 144.628,Z 351.551,A -85,B 0,C 180,E1 -29326.393,E2 -29326.393} C_VEL
LIN {X 0,Y 153.037,Z 342.763,A -85,B 0,C 180,E1 -29327.404,E2 -29327.404} C_VEL
LIN {X 0,Y 162.345,Z 331.163,A -85,B 0,C 180,E1 -29328.379,E2 -29328.379} C_VEL
LIN {X 0,Y 170.021,Z 319.565,A -85,B 0,C 180,E1 -29329.046,E2 -29329.046} C_VEL
LIN {X 0,Y 176.001,Z 308.588,A -85,B 0,C 180,E1 -29329.535,E2 -29329.535} C_VEL
LIN {X 0,Y 182.002,Z 294.774,A -85,B 0,C 180,E1 -29329.971,E2 -29329.971} C_VEL
LIN {X 0,Y 184.42,Z 287.896,A -85,B 0,C 180,E1 -29330.124,E2 -29330.124} C_VEL
LIN {X 0,Y 184.781,Z 286.768,A -85,B 0,C 180,E1 -29330.271,E2 -29330.271} C_VEL
LIN {X 0,Y 184.969,Z 285.772,A -85,B 0,C 180,E1 -29333.448,E2 -29333.448} C_VEL
LIN {X 0,Y 184.897,Z 286.204,A -85,B 0,C 180,E1 -29334.209,E2 -29334.209} C_VEL
LIN {X 0,Y 180.15,Z 299.219,A -85,B 0,C 180,E1 -29334.684,E2 -29334.684} C_VEL
LIN {X 0,Y 179.821,Z 299.97,A -85,B 0,C 180,E1 -29334.71,E2 -29334.71} C_VEL
LIN {X 0,Y 177.351,Z 305.47,A -85,B 0,C 180,E1 -29334.711,E2 -29334.711} C_VEL
LIN {X 0,Y 172.779,Z 314.183,A -85,B 0,C 180,E1 -29334.197,E2 -29334.197} C_VEL
LIN {X 0,Y 167.787,Z 322.508,A -85,B 0,C 180,E1 -29333.709,E2 -29333.709} C_VEL
LIN {X 0,Y 164.538,Z 327.32,A -85,B 0,C 180,E1 -29333.77,E2 -29333.77} C_VEL
LIN {X 0,Y 156.2,Z 338.21,A -85,B 0,C 180,E1 -29334.586,E2 -29334.586} C_VEL
LIN {X 0,Y 146.264,Z 348.96,A -85,B 0,C 180,E1 -29335.638,E2 -29335.638} C_VEL
LIN {X 0,Y 135.47,Z 358.571,A -85,B 0,C 180,E1 -29337.017,E2 -29337.017} C_VEL
LIN {X 0,Y 124.792,Z 366.481,A -85,B 0,C 180,E1 -29338.618,E2 -29338.618} C_VEL
LIN {X 0,Y 114.628,Z 372.789,A -85,B 0,C 180,E1 -29340.427,E2 -29340.427} C_VEL
LIN {X 0,Y 102.072,Z 379.11,A -85,B 0,C 180,E1 -29343.213,E2 -29343.213} C_VEL
LIN {X 0,Y 91.903,Z 383.223,A -85,B 0,C 180,E1 -29346.152,E2 -29346.152} C_VEL
LIN {X 0,Y 81.772,Z 386.412,A -85,B 0,C 180,E1 -29349.881,E2 -29349.881} C_VEL
LIN {X 0,Y 72.554,Z 388.597,A -85,B 0,C 180,E1 -29354.354,E2 -29354.354} C_VEL
LIN {X 0,Y 60.913,Z 390.273,A -85,B 0,C 180,E1 -29362.604,E2 -29362.604} C_VEL
LIN {X 0,Y 51.036,Z 390.498,A -85,B 0,C 180,E1 -29374.266,E2 -29374.266} C_VEL
LIN {X 0,Y 43.932,Z 389.29,A -85,B 0,C 180,E1 -29390.199,E2 -29390.199} C_VEL
LIN {X 0,Y 41.859,Z 388.147,A -85,B 0,C 180,E1 -29399.74,E2 -29399.74} C_VEL
LIN {X 0,Y 40.746,Z 386.652,A -85,B 0,C 180,E1 -29409.805,E2 -29409.805} C_VEL
LIN {X 0,Y 41.254,Z 383.666,A -85,B 0,C 180,E1 -29425.1,E2 -29425.1} C_VEL
LIN {X 0,Y 44.059,Z 379.846,A -85,B 0,C 180,E1 -29439.165,E2 -29439.165} C_VEL
LIN {X 0,Y 48.569,Z 375.136,A -85,B 0,C 180,E1 -29451.195,E2 -29451.195} C_VEL
LIN {X 0,Y 55.762,Z 368.285,A -85,B 0,C 180,E1 -29462.376,E2 -29462.376} C_VEL
LIN {X 0,Y 63.144,Z 361.127,A -85,B 0,C 180,E1 -29469.778,E2 -29469.778} C_VEL
LIN {X 0,Y 71.162,Z 352.541,A -85,B 0,C 180,E1 -29475.715,E2 -29475.715} C_VEL
LIN {X 0,Y 79.626,Z 342.167,A -85,B 0,C 180,E1 -29480.549,E2 -29480.549} C_VEL
LIN {X 0,Y 88.018,Z 330.468,A -85,B 0,C 180,E1 -29483.934,E2 -29483.934} C_VEL
LIN {X 0,Y 94.943,Z 318.824,A -85,B 0,C 180,E1 -29486.372,E2 -29486.372} C_VEL
LIN {X 0,Y 100.468,Z 307.773,A -85,B 0,C 180,E1 -29488.002,E2 -29488.002} C_VEL
LIN {X 0,Y 105.568,Z 295.035,A -85,B 0,C 180,E1 -29489.45,E2 -29489.45} C_VEL
LIN {X 0,Y 109.533,Z 282.179,A -85,B 0,C 180,E1 -29490.496,E2 -29490.496} C_VEL
LIN {X 0,Y 112.667,Z 267.935,A -85,B 0,C 180,E1 -29491.244,E2 -29491.244} C_VEL
LIN {X 0,Y 115.232,Z 248.679,A -85,B 0,C 180,E1 -29491.765,E2 -29491.765} C_VEL
LIN {X 0,Y 116.909,Z 233.65,A -85,B 0,C 180,E1 -29492.221,E2 -29492.221} C_VEL
LIN {X 0,Y 115.102,Z 228.224,A -85,B 0,C 180,E1 -29496.205,E2 -29496.205} C_VEL
LIN {X 0,Y 113.637,Z 224.312,A -85,B 0,C 180,E1 -29500.387,E2 -29500.387} C_VEL
LIN {X 0,Y 112.754,Z 221.8,A -85,B 0,C 180,E1 -29504.094,E2 -29504.094} C_VEL
LIN {X 0,Y 112.24,Z 218.251,A -85,B 0,C 180,E1 -29512.818,E2 -29512.818} C_VEL
LIN {X 0,Y 112.979,Z 222.012,A -85,B 0,C 180,E1 -29520.459,E2 -29520.459} C_VEL
LIN {X 0,Y 114.256,Z 225.698,A -85,B 0,C 180,E1 -29525.105,E2 -29525.105} C_VEL
LIN {X 0,Y 116.045,Z 230.944,A -85,B 0,C 180,E1 -29529.598,E2 -29529.598} C_VEL
LIN {X 0,Y 117.005,Z 233.957,A -85,B 0,C 180,E1 -29531.589,E2 -29531.589} C_VEL
LIN {X 0,Y 112.883,Z 268.571,A -85,B 0,C 180,E1 -29532.634,E2 -29532.634} C_VEL
LIN {X 0,Y 109.961,Z 282.424,A -85,B 0,C 180,E1 -29533.293,E2 -29533.293} C_VEL
LIN {X 0,Y 105.988,Z 295.464,A -85,B 0,C 180,E1 -29534.147,E2 -29534.147} C_VEL
LIN {X 0,Y 101.124,Z 307.861,A -85,B 0,C 180,E1 -29535.38,E2 -29535.38} C_VEL
LIN {X 0,Y 95.494,Z 319.402,A -85,B 0,C 180,E1 -29536.934,E2 -29536.934} C_VEL
LIN {X 0,Y 90.051,Z 328.869,A -85,B 0,C 180,E1 -29538.683,E2 -29538.683} C_VEL
LIN {X 0,Y 82.179,Z 340.438,A -85,B 0,C 180,E1 -29541.579,E2 -29541.579} C_VEL
LIN {X 0,Y 73.966,Z 350.79,A -85,B 0,C 180,E1 -29545.509,E2 -29545.509} C_VEL
LIN {X 0,Y 65.51,Z 360.14,A -85,B 0,C 180,E1 -29550.896,E2 -29550.896} C_VEL
LIN {X 0,Y 57.268,Z 368.314,A -85,B 0,C 180,E1 -29558.171,E2 -29558.171} C_VEL
LIN {X 0,Y 51.065,Z 374.355,A -85,B 0,C 180,E1 -29566.532,E2 -29566.532} C_VEL
LIN {X 0,Y 45.783,Z 379.626,A -85,B 0,C 180,E1 -29577.517,E2 -29577.517} C_VEL
LIN {X 0,Y 42.485,Z 383.903,A -85,B 0,C 180,E1 -29590.694,E2 -29590.694} C_VEL
LIN {X 0,Y 41.461,Z 386.233,A -85,B 0,C 180,E1 -29600.255,E2 -29600.255} C_VEL
LIN {X 0,Y 41.344,Z 388.165,A -85,B 0,C 180,E1 -29610.014,E2 -29610.014} C_VEL
LIN {X 0,Y 41.531,Z 389.687,A -85,B 0,C 180,E1 -29619.757,E2 -29619.757} C_VEL
LIN {X 0,Y 44.684,Z 391.692,A -85,B 0,C 180,E1 -29638.168,E2 -29638.168} C_VEL
LIN {X 0,Y 51.526,Z 392.404,A -85,B 0,C 180,E1 -29653.013,E2 -29653.013} C_VEL
LIN {X 0,Y 60.969,Z 391.849,A -85,B 0,C 180,E1 -29663.81,E2 -29663.81} C_VEL
LIN {X 0,Y 71.967,Z 390.021,A -85,B 0,C 180,E1 -29671.526,E2 -29671.526} C_VEL
LIN {X 0,Y 83.948,Z 386.878,A -85,B 0,C 180,E1 -29677.075,E2 -29677.075} C_VEL
LIN {X 0,Y 96.539,Z 382.33,A -85,B 0,C 180,E1 -29681.172,E2 -29681.172} C_VEL
LIN {X 0,Y 109.604,Z 376.187,A -85,B 0,C 180,E1 -29684.135,E2 -29684.135} C_VEL
LIN {X 0,Y 121.221,Z 369.379,A -85,B 0,C 180,E1 -29686.212,E2 -29686.212} C_VEL
LIN {X 0,Y 132.943,Z 360.982,A -85,B 0,C 180,E1 -29687.979,E2 -29687.979} C_VEL
LIN {X 0,Y 143.131,Z 352.239,A -85,B 0,C 180,E1 -29689.144,E2 -29689.144} C_VEL
LIN {X 0,Y 151.657,Z 343.624,A -85,B 0,C 180,E1 -29690.002,E2 -29690.002} C_VEL
LIN {X 0,Y 161.076,Z 332.236,A -85,B 0,C 180,E1 -29690.829,E2 -29690.829} C_VEL
LIN {X 0,Y 169.689,Z 319.498,A -85,B 0,C 180,E1 -29691.447,E2 -29691.447} C_VEL
LIN {X 0,Y 176.236,Z 307.522,A -85,B 0,C 180,E1 -29691.869,E2 -29691.869} C_VEL
LIN {X 0,Y 179.358,Z 300.746,A -85,B 0,C 180,E1 -29692.066,E2 -29692.066} C_VEL
LIN {X 0,Y 180.062,Z 299.119,A -85,B 0,C 180,E1 -29692.417,E2 -29692.417} C_VEL
LIN {X 0,Y 174.567,Z 310.825,A -85,B 0,C 180,E1 -29692.88,E2 -29692.88} C_VEL
LIN {X 0,Y 167.105,Z 323.526,A -85,B 0,C 180,E1 -29693.543,E2 -29693.543} C_VEL
LIN {X 0,Y 164.538,Z 327.32,A -85,B 0,C 180,E1 -29693.77,E2 -29693.77} C_VEL
LIN {X 0,Y 160.725,Z 332.655,A -85,B 0,C 180,E1 -29693.889,E2 -29693.889} C_VEL
LIN {X 0,Y 153.789,Z 341.121,A -85,B 0,C 180,E1 -29693.516,E2 -29693.516} C_VEL
LIN {X 0,Y 146.21,Z 348.998,A -85,B 0,C 180,E1 -29693.138,E2 -29693.138} C_VEL
LIN {X 0,Y 141.378,Z 353.406,A -85,B 0,C 180,E1 -29693.302,E2 -29693.302} C_VEL
LIN {X 0,Y 130.632,Z 362.155,A -85,B 0,C 180,E1 -29694.484,E2 -29694.484} C_VEL
LIN {X 0,Y 119.791,Z 369.477,A -85,B 0,C 180,E1 -29695.908,E2 -29695.908} C_VEL
LIN {X 0,Y 109.035,Z 375.48,A -85,B 0,C 180,E1 -29697.647,E2 -29697.647} C_VEL
LIN {X 0,Y 97.291,Z 380.816,A -85,B 0,C 180,E1 -29699.986,E2 -29699.986} C_VEL
LIN {X 0,Y 84.494,Z 385.321,A -85,B 0,C 180,E1 -29703.396,E2 -29703.396} C_VEL
LIN {X 0,Y 77.7,Z 387.181,A -85,B 0,C 180,E1 -29705.686,E2 -29705.686} C_VEL
LIN {X 0,Y 64.607,Z 389.703,A -85,B 0,C 180,E1 -29711.714,E2 -29711.714} C_VEL
LIN {X 0,Y 52.572,Z 390.749,A -85,B 0,C 180,E1 -29720.614,E2 -29720.614} C_VEL
LIN {X 0,Y 42.41,Z 390.354,A -85,B 0,C 180,E1 -29734.023,E2 -29734.023} C_VEL
LIN {X 0,Y 35.618,Z 388.523,A -85,B 0,C 180,E1 -29753.685,E2 -29753.685} C_VEL
LIN {X 0,Y 33.909,Z 387.075,A -85,B 0,C 180,E1 -29765.492,E2 -29765.492} C_VEL
LIN {X 0,Y 34.691,Z 383.067,A -85,B 0,C 180,E1 -29789.983,E2 -29789.983} C_VEL
LIN {X 0,Y 38.413,Z 379.005,A -85,B 0,C 180,E1 -29805.913,E2 -29805.913} C_VEL
LIN {X 0,Y 43.99,Z 374.03,A -85,B 0,C 180,E1 -29818.624,E2 -29818.624} C_VEL
LIN {X 0,Y 52.445,Z 366.866,A -85,B 0,C 180,E1 -29829.52,E2 -29829.52} C_VEL
LIN {X 0,Y 60.981,Z 359.07,A -85,B 0,C 180,E1 -29836.606,E2 -29836.606} C_VEL
LIN {X 0,Y 69.384,Z 350.4,A -85,B 0,C 180,E1 -29841.708,E2 -29841.708} C_VEL
LIN {X 0,Y 76.842,Z 341.532,A -85,B 0,C 180,E1 -29845.387,E2 -29845.387} C_VEL
LIN {X 0,Y 84.815,Z 330.844,A -85,B 0,C 180,E1 -29848.127,E2 -29848.127} C_VEL
LIN {X 0,Y 91.999,Z 319.24,A -85,B 0,C 180,E1 -29850.325,E2 -29850.325} C_VEL
LIN {X 0,Y 97.708,Z 308.235,A -85,B 0,C 180,E1 -29851.766,E2 -29851.766} C_VEL
LIN {X 0,Y 102.95,Z 295.599,A -85,B 0,C 180,E1 -29853.068,E2 -29853.068} C_VEL
LIN {X 0,Y 107.133,Z 282.485,A -85,B 0,C 180,E1 -29854.026,E2 -29854.026} C_VEL
LIN {X 0,Y 110.339,Z 268.357,A -85,B 0,C 180,E1 -29854.685,E2 -29854.685} C_VEL
LIN {X 0,Y 113.113,Z 247.846,A -85,B 0,C 180,E1 -29855.188,E2 -29855.188} C_VEL
LIN {X 0,Y 114.33,Z 237.288,A -85,B 0,C 180,E1 -29855.474,E2 -29855.474} C_VEL
LIN {X 0,Y 113.087,Z 233.109,A -85,B 0,C 180,E1 -29858.994,E2 -29858.994} C_VEL
LIN {X 0,Y 112.058,Z 230.041,A -85,B 0,C 180,E1 -29862.837,E2 -29862.837} C_VEL
LIN {X 0,Y 111.6,Z 228.459,A -85,B 0,C 180,E1 -29865.423,E2 -29865.423} C_VEL
LIN {X 0,Y 111.326,Z 225.523,A -85,B 0,C 180,E1 -29872.759,E2 -29872.759} C_VEL
LIN {X 0,Y 111.873,Z 228.848,A -85,B 0,C 180,E1 -29879.595,E2 -29879.595} C_VEL
LIN {X 0,Y 112.971,Z 232.485,A -85,B 0,C 180,E1 -29884.178,E2 -29884.178} C_VEL
LIN {X 0,Y 114.414,Z 237.528,A -85,B 0,C 180,E1 -29888.347,E2 -29888.347} C_VEL
LIN {X 0,Y 110.516,Z 268.914,A -85,B 0,C 180,E1 -29889.212,E2 -29889.212} C_VEL
LIN {X 0,Y 107.505,Z 282.648,A -85,B 0,C 180,E1 -29889.792,E2 -29889.792} C_VEL
LIN {X 0,Y 103.212,Z 296.215,A -85,B 0,C 180,E1 -29890.585,E2 -29890.585} C_VEL
LIN {X 0,Y 97.805,Z 309.308,A -85,B 0,C 180,E1 -29891.778,E2 -29891.778} C_VEL
LIN {X 0,Y 91.543,Z 321.336,A -85,B 0,C 180,E1 -29893.257,E2 -29893.257} C_VEL
LIN {X 0,Y 86.302,Z 329.973,A -85,B 0,C 180,E1 -29894.779,E2 -29894.779} C_VEL
LIN {X 0,Y 79.015,Z 340.151,A -85,B 0,C 180,E1 -29897.054,E2 -29897.054} C_VEL
LIN {X 0,Y 71.168,Z 349.663,A -85,B 0,C 180,E1 -29900.281,E2 -29900.281} C_VEL
LIN {X 0,Y 62.128,Z 359.192,A -85,B 0,C 180,E1 -29905.204,E2 -29905.204} C_VEL
LIN {X 0,Y 53.997,Z 366.789,A -85,B 0,C 180,E1 -29911.401,E2 -29911.401} C_VEL
LIN {X 0,Y 46.116,Z 373.608,A -85,B 0,C 180,E1 -29920.38,E2 -29920.38} C_VEL
LIN {X 0,Y 39.938,Z 378.986,A -85,B 0,C 180,E1 -29932.001,E2 -29932.001} C_VEL
LIN {X 0,Y 35.814,Z 383.365,A -85,B 0,C 180,E1 -29946.909,E2 -29946.909} C_VEL
LIN {X 0,Y 34.476,Z 385.746,A -85,B 0,C 180,E1 -29958.255,E2 -29958.255} C_VEL
LIN {X 0,Y 34.259,Z 387.727,A -85,B 0,C 180,E1 -29970.017,E2 -29970.017} C_VEL
LIN {X 0,Y 34.556,Z 389.293,A -85,B 0,C 180,E1 -29981.752,E2 -29981.752} C_VEL
LIN {X 0,Y 38.548,Z 391.386,A -85,B 0,C 180,E1 -30003.176,E2 -30003.176} C_VEL
LIN {X 0,Y 46.564,Z 392.186,A -85,B 0,C 180,E1 -30019.015,E2 -30019.015} C_VEL
LIN {X 0,Y 57.043,Z 391.719,A -85,B 0,C 180,E1 -30029.61,E2 -30029.61} C_VEL
LIN {X 0,Y 68.847,Z 389.978,A -85,B 0,C 180,E1 -30036.762,E2 -30036.762} C_VEL
LIN {X 0,Y 81.434,Z 386.927,A -85,B 0,C 180,E1 -30041.704,E2 -30041.704} C_VEL
LIN {X 0,Y 94.484,Z 382.477,A -85,B 0,C 180,E1 -30045.257,E2 -30045.257} C_VEL
LIN {X 0,Y 107.881,Z 376.482,A -85,B 0,C 180,E1 -30047.761,E2 -30047.761} C_VEL
LIN {X 0,Y 119.732,Z 369.79,A -85,B 0,C 180,E1 -30049.504,E2 -30049.504} C_VEL
LIN {X 0,Y 131.654,Z 361.522,A -85,B 0,C 180,E1 -30050.983,E2 -30050.983} C_VEL
LIN {X 0,Y 141.97,Z 352.928,A -85,B 0,C 180,E1 -30051.944,E2 -30051.944} C_VEL
LIN {X 0,Y 148.851,Z 346.241,A -85,B 0,C 180,E1 -30052.559,E2 -30052.559} C_VEL
LIN {X 0,Y 141.378,Z 353.406,A -85,B 0,C 180,E1 -30053.302,E2 -30053.302} C_VEL
LIN {X 0,Y 137.297,Z 356.9,A -85,B 0,C 180,E1 -30053.549,E2 -30053.549} C_VEL
LIN {X 0,Y 128.786,Z 363.465,A -85,B 0,C 180,E1 -30053.612,E2 -30053.612} C_VEL
LIN {X 0,Y 119.873,Z 369.431,A -85,B 0,C 180,E1 -30053.484,E2 -30053.484} C_VEL
LIN {X 0,Y 115.269,Z 372.153,A -85,B 0,C 180,E1 -30053.52,E2 -30053.52} C_VEL
LIN {X 0,Y 108.236,Z 375.85,A -85,B 0,C 180,E1 -30053.944,E2 -30053.944} C_VEL
LIN {X 0,Y 105.88,Z 376.965,A -85,B 0,C 180,E1 -30054.238,E2 -30054.238} C_VEL
LIN {X 0,Y 96.141,Z 381.176,A -85,B 0,C 180,E1 -30055.794,E2 -30055.794} C_VEL
LIN {X 0,Y 84.384,Z 385.2,A -85,B 0,C 180,E1 -30058.258,E2 -30058.258} C_VEL
LIN {X 0,Y 70.346,Z 388.649,A -85,B 0,C 180,E1 -30062.294,E2 -30062.294} C_VEL
LIN {X 0,Y 56.834,Z 390.542,A -85,B 0,C 180,E1 -30068.335,E2 -30068.335} C_VEL
LIN {X 0,Y 44.311,Z 390.964,A -85,B 0,C 180,E1 -30077.852,E2 -30077.852} C_VEL
LIN {X 0,Y 33.778,Z 389.949,A -85,B 0,C 180,E1 -30093.639,E2 -30093.639} C_VEL
LIN {X 0,Y 29.919,Z 388.9,A -85,B 0,C 180,E1 -30105.168,E2 -30105.168} C_VEL
LIN {X 0,Y 27.333,Z 387.499,A -85,B 0,C 180,E1 -30119.028,E2 -30119.028} C_VEL
LIN {X 0,Y 27.361,Z 383.595,A -85,B 0,C 180,E1 -30149.979,E2 -30149.979} C_VEL
LIN {X 0,Y 31.53,Z 379.623,A -85,B 0,C 180,E1 -30169.513,E2 -30169.513} C_VEL
LIN {X 0,Y 37.85,Z 374.757,A -85,B 0,C 180,E1 -30183.833,E2 -30183.833} C_VEL
LIN {X 0,Y 47.151,Z 367.713,A -85,B 0,C 180,E1 -30195.056,E2 -30195.056} C_VEL
LIN {X 0,Y 57.497,Z 358.992,A -85,B 0,C 180,E1 -30202.598,E2 -30202.598} C_VEL
LIN {X 0,Y 66.77,Z 349.905,A -85,B 0,C 180,E1 -30207.342,E2 -30207.342} C_VEL
LIN {X 0,Y 74.649,Z 340.895,A -85,B 0,C 180,E1 -30210.542,E2 -30210.542} C_VEL
LIN {X 0,Y 82.906,Z 330.048,A -85,B 0,C 180,E1 -30212.869,E2 -30212.869} C_VEL
LIN {X 0,Y 90.353,Z 318.222,A -85,B 0,C 180,E1 -30214.705,E2 -30214.705} C_VEL
LIN {X 0,Y 96.206,Z 306.944,A -85,B 0,C 180,E1 -30215.928,E2 -30215.928} C_VEL
LIN {X 0,Y 101.605,Z 293.875,A -85,B 0,C 180,E1 -30217.032,E2 -30217.032} C_VEL
LIN {X 0,Y 105.346,Z 282.085,A -85,B 0,C 180,E1 -30217.752,E2 -30217.752} C_VEL
LIN {X 0,Y 108.432,Z 268.738,A -85,B 0,C 180,E1 -30218.264,E2 -30218.264} C_VEL
LIN {X 0,Y 111.234,Z 248.593,A -85,B 0,C 180,E1 -30218.669,E2 -30218.669} C_VEL
LIN {X 0,Y 112.098,Z 241.059,A -85,B 0,C 180,E1 -30218.913,E2 -30218.913} C_VEL
LIN {X 0,Y 111.059,Z 237.244,A -85,B 0,C 180,E1 -30223.12,E2 -30223.12} C_VEL
LIN {X 0,Y 110.579,Z 235.311,A -85,B 0,C 180,E1 -30226.212,E2 -30226.212} C_VEL
LIN {X 0,Y 110.409,Z 232.816,A -85,B 0,C 180,E1 -30232.698,E2 -30232.698} C_VEL
LIN {X 0,Y 110.761,Z 235.57,A -85,B 0,C 180,E1 -30238.505,E2 -30238.505} C_VEL
LIN {X 0,Y 111.554,Z 238.759,A -85,B 0,C 180,E1 -30242.624,E2 -30242.624} C_VEL
LIN {X 0,Y 112.176,Z 241.399,A -85,B 0,C 180,E1 -30244.987,E2 -30244.987} C_VEL
LIN {X 0,Y 108.608,Z 268.971,A -85,B 0,C 180,E1 -30245.636,E2 -30245.636} C_VEL
LIN {X 0,Y 105.361,Z 283.278,A -85,B 0,C 180,E1 -30246.171,E2 -30246.171} C_VEL
LIN {X 0,Y 100.855,Z 296.963,A -85,B 0,C 180,E1 -30246.835,E2 -30246.835} C_VEL
LIN {X 0,Y 95.745,Z 308.956,A -85,B 0,C 180,E1 -30247.762,E2 -30247.762} C_VEL
LIN {X 0,Y 89.392,Z 320.892,A -85,B 0,C 180,E1 -30248.971,E2 -30248.971} C_VEL
LIN {X 0,Y 83.913,Z 329.669,A -85,B 0,C 180,E1 -30250.271,E2 -30250.271} C_VEL
LIN {X 0,Y 76.385,Z 339.864,A -85,B 0,C 180,E1 -30252.194,E2 -30252.194} C_VEL
LIN {X 0,Y 67.386,Z 350.255,A -85,B 0,C 180,E1 -30255.298,E2 -30255.298} C_VEL
LIN {X 0,Y 57.867,Z 359.63,A -85,B 0,C 180,E1 -30259.768,E2 -30259.768} C_VEL
LIN {X 0,Y 49.782,Z 366.626,A -85,B 0,C 180,E1 -30265.086,E2 -30265.086} C_VEL
LIN {X 0,Y 41.829,Z 372.855,A -85,B 0,C 180,E1 -30272.877,E2 -30272.877} C_VEL
LIN {X 0,Y 34.591,Z 378.346,A -85,B 0,C 180,E1 -30284.698,E2 -30284.698} C_VEL
LIN {X 0,Y 28.274,Z 384.084,A -85,B 0,C 180,E1 -30308.13,E2 -30308.13} C_VEL
LIN {X 0,Y 27.147,Z 387.287,A -85,B 0,C 180,E1 -30330.021,E2 -30330.021} C_VEL
LIN {X 0,Y 27.633,Z 388.899,A -85,B 0,C 180,E1 -30344.755,E2 -30344.755} C_VEL
LIN {X 0,Y 32.819,Z 391.08,A -85,B 0,C 180,E1 -30369.996,E2 -30369.996} C_VEL
LIN {X 0,Y 42.231,Z 391.967,A -85,B 0,C 180,E1 -30386.339,E2 -30386.339} C_VEL
LIN {X 0,Y 53.777,Z 391.587,A -85,B 0,C 180,E1 -30396.204,E2 -30396.204} C_VEL
LIN {X 0,Y 66.356,Z 389.936,A -85,B 0,C 180,E1 -30402.432,E2 -30402.432} C_VEL
LIN {X 0,Y 79.485,Z 386.975,A -85,B 0,C 180,E1 -30406.588,E2 -30406.588} C_VEL
LIN {X 0,Y 92.931,Z 382.62,A -85,B 0,C 180,E1 -30409.496,E2 -30409.496} C_VEL
LIN {X 0,Y 106.602,Z 376.74,A -85,B 0,C 180,E1 -30411.495,E2 -30411.495} C_VEL
LIN {X 0,Y 113.473,Z 373.168,A -85,B 0,C 180,E1 -30412.326,E2 -30412.326} C_VEL
LIN {X 0,Y 115.091,Z 372.211,A -85,B 0,C 180,E1 -30412.974,E2 -30412.974} C_VEL
LIN {X 0,Y 105.88,Z 376.965,A -85,B 0,C 180,E1 -30414.238,E2 -30414.238} C_VEL
LIN {X 0,Y 100.372,Z 379.454,A -85,B 0,C 180,E1 -30414.699,E2 -30414.699} C_VEL
LIN {X 0,Y 90.877,Z 383.119,A -85,B 0,C 180,E1 -30414.507,E2 -30414.507} C_VEL
LIN {X 0,Y 81.184,Z 386.167,A -85,B 0,C 180,E1 -30414.314,E2 -30414.314} C_VEL
LIN {X 0,Y 75.369,Z 387.583,A -85,B 0,C 180,E1 -30415,E2 -30415} C_VEL
LIN {X 0,Y 63.294,Z 389.835,A -85,B 0,C 180,E1 -30418.156,E2 -30418.156} C_VEL
LIN {X 0,Y 49.319,Z 391.116,A -85,B 0,C 180,E1 -30423.89,E2 -30423.89} C_VEL
LIN {X 0,Y 36.193,Z 390.918,A -85,B 0,C 180,E1 -30433.788,E2 -30433.788} C_VEL
LIN {X 0,Y 25.154,Z 389.279,A -85,B 0,C 180,E1 -30453.007,E2 -30453.007} C_VEL
LIN {X 0,Y 21.318,Z 387.922,A -85,B 0,C 180,E1 -30468.714,E2 -30468.714} C_VEL
LIN {X 0,Y 19.393,Z 385.227,A -85,B 0,C 180,E1 -30499.53,E2 -30499.53} C_VEL
LIN {X 0,Y 22.876,Z 381.64,A -85,B 0,C 180,E1 -30527.866,E2 -30527.866} C_VEL
LIN {X 0,Y 29.539,Z 377.155,A -85,B 0,C 180,E1 -30546.475,E2 -30546.475} C_VEL
LIN {X 0,Y 39.338,Z 370.679,A -85,B 0,C 180,E1 -30559.378,E2 -30559.378} C_VEL
LIN {X 0,Y 50.24,Z 362.628,A -85,B 0,C 180,E1 -30567.047,E2 -30567.047} C_VEL
LIN {X 0,Y 58.717,Z 355.313,A -85,B 0,C 180,E1 -30571.16,E2 -30571.16} C_VEL
LIN {X 0,Y 66.466,Z 347.713,A -85,B 0,C 180,E1 -30573.977,E2 -30573.977} C_VEL
LIN {X 0,Y 74.827,Z 338.233,A -85,B 0,C 180,E1 -30576.293,E2 -30576.293} C_VEL
LIN {X 0,Y 83.271,Z 326.792,A -85,B 0,C 180,E1 -30578.165,E2 -30578.165} C_VEL
LIN {X 0,Y 91.008,Z 314.059,A -85,B 0,C 180,E1 -30579.427,E2 -30579.427} C_VEL
LIN {X 0,Y 96.96,Z 301.79,A -85,B 0,C 180,E1 -30580.42,E2 -30580.42} C_VEL
LIN {X 0,Y 102.049,Z 288.288,A -85,B 0,C 180,E1 -30581.234,E2 -30581.234} C_VEL
LIN {X 0,Y 105.532,Z 275.825,A -85,B 0,C 180,E1 -30581.767,E2 -30581.767} C_VEL
LIN {X 0,Y 108.101,Z 262.373,A -85,B 0,C 180,E1 -30582.081,E2 -30582.081} C_VEL
LIN {X 0,Y 110.233,Z 245.411,A -85,B 0,C 180,E1 -30582.407,E2 -30582.407} C_VEL
LIN {X 0,Y 109.631,Z 242.347,A -85,B 0,C 180,E1 -30586.556,E2 -30586.556} C_VEL
LIN {X 0,Y 109.503,Z 240.025,A -85,B 0,C 180,E1 -30592.637,E2 -30592.637} C_VEL
LIN {X 0,Y 109.703,Z 242.322,A -85,B 0,C 180,E1 -30597.488,E2 -30597.488} C_VEL
LIN {X 0,Y 110.269,Z 245.327,A -85,B 0,C 180,E1 -30601.306,E2 -30601.306} C_VEL
LIN {X 0,Y 110.294,Z 245.497,A -85,B 0,C 180,E1 -30601.453,E2 -30601.453} C_VEL
LIN {X 0,Y 107.185,Z 268.779,A -85,B 0,C 180,E1 -30601.942,E2 -30601.942} C_VEL
LIN {X 0,Y 103.887,Z 283.056,A -85,B 0,C 180,E1 -30602.363,E2 -30602.363} C_VEL
LIN {X 0,Y 99.36,Z 296.619,A -85,B 0,C 180,E1 -30602.857,E2 -30602.857} C_VEL
LIN {X 0,Y 94.174,Z 308.604,A -85,B 0,C 180,E1 -30603.592,E2 -30603.592} C_VEL
LIN {X 0,Y 87.76,Z 320.459,A -85,B 0,C 180,E1 -30604.511,E2 -30604.511} C_VEL
LIN {X 0,Y 82.072,Z 329.365,A -85,B 0,C 180,E1 -30605.528,E2 -30605.528} C_VEL
LIN {X 0,Y 74.34,Z 339.574,A -85,B 0,C 180,E1 -30607.018,E2 -30607.018} C_VEL
LIN {X 0,Y 65.856,Z 349.114,A -85,B 0,C 180,E1 -30609.258,E2 -30609.258} C_VEL
LIN {X 0,Y 55.843,Z 358.674,A -85,B 0,C 180,E1 -30612.795,E2 -30612.795} C_VEL
LIN {X 0,Y 46.427,Z 366.354,A -85,B 0,C 180,E1 -30617.652,E2 -30617.652} C_VEL
LIN {X 0,Y 35.483,Z 374.119,A -85,B 0,C 180,E1 -30626.999,E2 -30626.999} C_VEL
LIN {X 0,Y 27.482,Z 379.341,A -85,B 0,C 180,E1 -30639.932,E2 -30639.932} C_VEL
LIN {X 0,Y 21.817,Z 383.547,A -85,B 0,C 180,E1 -30661.136,E2 -30661.136} C_VEL
LIN {X 0,Y 20.039,Z 386.847,A -85,B 0,C 180,E1 -30690.029,E2 -30690.029} C_VEL
LIN {X 0,Y 20.848,Z 388.505,A -85,B 0,C 180,E1 -30709.73,E2 -30709.73} C_VEL
LIN {X 0,Y 27.733,Z 390.773,A -85,B 0,C 180,E1 -30739.517,E2 -30739.517} C_VEL
LIN {X 0,Y 38.737,Z 391.749,A -85,B 0,C 180,E1 -30755.148,E2 -30755.148} C_VEL
LIN {X 0,Y 51.311,Z 391.456,A -85,B 0,C 180,E1 -30763.53,E2 -30763.53} C_VEL
LIN {X 0,Y 64.562,Z 389.893,A -85,B 0,C 180,E1 -30768.483,E2 -30768.483} C_VEL
LIN {X 0,Y 78.141,Z 387.023,A -85,B 0,C 180,E1 -30771.674,E2 -30771.674} C_VEL
LIN {X 0,Y 85.003,Z 385.074,A -85,B 0,C 180,E1 -30772.866,E2 -30772.866} C_VEL
LIN {X 0,Y 84.954,Z 385.08,A -85,B 0,C 180,E1 -30773.138,E2 -30773.138} C_VEL
LIN {X 0,Y 75.369,Z 387.583,A -85,B 0,C 180,E1 -30775,E2 -30775} C_VEL
LIN {X 0,Y 69.452,Z 388.847,A -85,B 0,C 180,E1 -30775.825,E2 -30775.825} C_VEL
LIN {X 0,Y 59.299,Z 390.38,A -85,B 0,C 180,E1 -30775.877,E2 -30775.877} C_VEL
LIN {X 0,Y 51.121,Z 391.131,A -85,B 0,C 180,E1 -30775.82,E2 -30775.82} C_VEL
LIN {X 0,Y 45.065,Z 391.371,A -85,B 0,C 180,E1 -30776.778,E2 -30776.778} C_VEL
LIN {X 0,Y 43.106,Z 391.4,A -85,B 0,C 180,E1 -30777.504,E2 -30777.504} C_VEL
LIN {X 0,Y 35.166,Z 391.199,A -85,B 0,C 180,E1 -30781.744,E2 -30781.744} C_VEL
LIN {X 0,Y 21.975,Z 389.66,A -85,B 0,C 180,E1 -30796.278,E2 -30796.278} C_VEL
LIN {X 0,Y 16.461,Z 388.349,A -85,B 0,C 180,E1 -30811.298,E2 -30811.298} C_VEL
LIN {X 0,Y 12.221,Z 385.737,A -85,B 0,C 180,E1 -30853.24,E2 -30853.24} C_VEL
LIN {X 0,Y 16.094,Z 382.209,A -85,B 0,C 180,E1 -30895.852,E2 -30895.852} C_VEL
LIN {X 0,Y 24.154,Z 377.823,A -85,B 0,C 180,E1 -30916.635,E2 -30916.635} C_VEL
LIN {X 0,Y 35.107,Z 371.463,A -85,B 0,C 180,E1 -30928.266,E2 -30928.266} C_VEL
LIN {X 0,Y 46.738,Z 363.542,A -85,B 0,C 180,E1 -30934.422,E2 -30934.422} C_VEL
LIN {X 0,Y 55.646,Z 356.367,A -85,B 0,C 180,E1 -30937.567,E2 -30937.567} C_VEL
LIN {X 0,Y 65.365,Z 347.154,A -85,B 0,C 180,E1 -30940.158,E2 -30940.158} C_VEL
LIN {X 0,Y 73.121,Z 338.591,A -85,B 0,C 180,E1 -30941.62,E2 -30941.62} C_VEL
LIN {X 0,Y 81.758,Z 327.188,A -85,B 0,C 180,E1 -30942.977,E2 -30942.977} C_VEL
LIN {X 0,Y 89.621,Z 314.503,A -85,B 0,C 180,E1 -30943.847,E2 -30943.847} C_VEL
LIN {X 0,Y 95.682,Z 302.293,A -85,B 0,C 180,E1 -30944.568,E2 -30944.568} C_VEL
LIN {X 0,Y 100.854,Z 288.893,A -85,B 0,C 180,E1 -30945.19,E2 -30945.19} C_VEL
LIN {X 0,Y 104.416,Z 276.51,A -85,B 0,C 180,E1 -30945.586,E2 -30945.586} C_VEL
LIN {X 0,Y 107.191,Z 262.195,A -85,B 0,C 180,E1 -30945.821,E2 -30945.821} C_VEL
LIN {X 0,Y 108.74,Z 250.172,A -85,B 0,C 180,E1 -30946.006,E2 -30946.006} C_VEL
LIN {X 0,Y 108.599,Z 249.031,A -85,B 0,C 180,E1 -30947.858,E2 -30947.858} C_VEL
LIN {X 0,Y 108.591,Z 247.264,A -85,B 0,C 180,E1 -30952.575,E2 -30952.575} C_VEL
LIN {X 0,Y 108.686,Z 249.153,A -85,B 0,C 180,E1 -30956.552,E2 -30956.552} C_VEL
LIN {X 0,Y 108.8,Z 250.104,A -85,B 0,C 180,E1 -30957.912,E2 -30957.912} C_VEL
LIN {X 0,Y 106.043,Z 269.515,A -85,B 0,C 180,E1 -30958.192,E2 -30958.192} C_VEL
LIN {X 0,Y 102.505,Z 284.16,A -85,B 0,C 180,E1 -30958.502,E2 -30958.502} C_VEL
LIN {X 0,Y 97.963,Z 297.307,A -85,B 0,C 180,E1 -30958.827,E2 -30958.827} C_VEL
LIN {X 0,Y 92.237,Z 310.053,A -85,B 0,C 180,E1 -30959.41,E2 -30959.41} C_VEL
LIN {X 0,Y 85.467,Z 322.011,A -85,B 0,C 180,E1 -30960.015,E2 -30960.015} C_VEL
LIN {X 0,Y 77.309,Z 333.816,A -85,B 0,C 180,E1 -30960.993,E2 -30960.993} C_VEL
LIN {X 0,Y 68.573,Z 344.287,A -85,B 0,C 180,E1 -30962.404,E2 -30962.404} C_VEL
LIN {X 0,Y 58.153,Z 354.638,A -85,B 0,C 180,E1 -30964.533,E2 -30964.533} C_VEL
LIN {X 0,Y 47.686,Z 363.328,A -85,B 0,C 180,E1 -30967.73,E2 -30967.73} C_VEL
LIN {X 0,Y 36.117,Z 371.351,A -85,B 0,C 180,E1 -30973.425,E2 -30973.425} C_VEL
LIN {X 0,Y 26.542,Z 377.062,A -85,B 0,C 180,E1 -30982.122,E2 -30982.122} C_VEL
LIN {X 0,Y 15.939,Z 383.01,A -85,B 0,C 180,E1 -31008.64,E2 -31008.64} C_VEL
LIN {X 0,Y 12.945,Z 386.405,A -85,B 0,C 180,E1 -31050.044,E2 -31050.044} C_VEL
LIN {X 0,Y 14.351,Z 388.111,A -85,B 0,C 180,E1 -31079.367,E2 -31079.367} C_VEL
LIN {X 0,Y 23.733,Z 390.467,A -85,B 0,C 180,E1 -31112.724,E2 -31112.724} C_VEL
LIN {X 0,Y 36.323,Z 391.531,A -85,B 0,C 180,E1 -31125.398,E2 -31125.398} C_VEL
LIN {X 0,Y 49.76,Z 391.325,A -85,B 0,C 180,E1 -31131.44,E2 -31131.44} C_VEL
LIN {X 0,Y 52.621,Z 391.107,A -85,B 0,C 180,E1 -31132.3,E2 -31132.3} C_VEL
LIN {X 0,Y 49.388,Z 391.268,A -85,B 0,C 180,E1 -31135.069,E2 -31135.069} C_VEL
LIN {X 0,Y 43.106,Z 391.4,A -85,B 0,C 180,E1 -31137.504,E2 -31137.504} C_VEL
LIN {X 0,Y 37.353,Z 391.38,A -85,B 0,C 180,E1 -31139.389,E2 -31139.389} C_VEL
LIN {X 0,Y 27.481,Z 390.764,A -85,B 0,C 180,E1 -31140.455,E2 -31140.455} C_VEL
LIN {X 0,Y 19.569,Z 389.752,A -85,B 0,C 180,E1 -31141.277,E2 -31141.277} C_VEL
LIN {X 0,Y 13.826,Z 388.705,A -85,B 0,C 180,E1 -31145.217,E2 -31145.217} C_VEL
LIN {X 0,Y 12.026,Z 388.274,A -85,B 0,C 180,E1 -31148.421,E2 -31148.421} C_VEL
LIN {X 0,Y 5.314,Z 385.158,A -85,B 0,C 180,E1 -31229.892,E2 -31229.892} C_VEL
LIN {X 0,Y 13.234,Z 381.478,A -85,B 0,C 180,E1 -31282.734,E2 -31282.734} C_VEL
LIN {X 0,Y 23.3,Z 376.851,A -85,B 0,C 180,E1 -31294.749,E2 -31294.749} C_VEL
LIN {X 0,Y 35.392,Z 370.205,A -85,B 0,C 180,E1 -31300.554,E2 -31300.554} C_VEL
LIN {X 0,Y 47.625,Z 361.945,A -85,B 0,C 180,E1 -31303.533,E2 -31303.533} C_VEL
LIN {X 0,Y 58.083,Z 353.331,A -85,B 0,C 180,E1 -31305.423,E2 -31305.423} C_VEL
LIN {X 0,Y 68.535,Z 342.915,A -85,B 0,C 180,E1 -31306.913,E2 -31306.913} C_VEL
LIN {X 0,Y 77.355,Z 332.35,A -85,B 0,C 180,E1 -31307.564,E2 -31307.564} C_VEL
LIN {X 0,Y 85.245,Z 320.903,A -85,B 0,C 180,E1 -31308.211,E2 -31308.211} C_VEL
LIN {X 0,Y 92.285,Z 308.334,A -85,B 0,C 180,E1 -31308.633,E2 -31308.633} C_VEL
LIN {X 0,Y 98.394,Z 294.383,A -85,B 0,C 180,E1 -31309.116,E2 -31309.116} C_VEL
LIN {X 0,Y 102.449,Z 282.133,A -85,B 0,C 180,E1 -31309.417,E2 -31309.417} C_VEL
LIN {X 0,Y 105.665,Z 268.527,A -85,B 0,C 180,E1 -31309.589,E2 -31309.589} C_VEL
LIN {X 0,Y 107.525,Z 256.245,A -85,B 0,C 180,E1 -31309.633,E2 -31309.633} C_VEL
LIN {X 0,Y 107.61,Z 255.512,A -85,B 0,C 180,E1 -31309.748,E2 -31309.748} C_VEL
LIN {X 0,Y 107.682,Z 254.487,A -85,B 0,C 180,E1 -31312.512,E2 -31312.512} C_VEL
LIN {X 0,Y 107.67,Z 255.16,A -85,B 0,C 180,E1 -31314.198,E2 -31314.198} C_VEL
LIN {X 0,Y 105.043,Z 271.89,A -85,B 0,C 180,E1 -31314.377,E2 -31314.377} C_VEL
LIN {X 0,Y 101.554,Z 285.432,A -85,B 0,C 180,E1 -31314.58,E2 -31314.58} C_VEL
LIN {X 0,Y 97.037,Z 298.062,A -85,B 0,C 180,E1 -31314.713,E2 -31314.713} C_VEL
LIN {X 0,Y 90.722,Z 311.633,A -85,B 0,C 180,E1 -31315.074,E2 -31315.074} C_VEL
LIN {X 0,Y 83.666,Z 323.597,A -85,B 0,C 180,E1 -31315.296,E2 -31315.296} C_VEL
LIN {X 0,Y 76.631,Z 333.517,A -85,B 0,C 180,E1 -31315.739,E2 -31315.739} C_VEL
LIN {X 0,Y 68.65,Z 343.008,A -85,B 0,C 180,E1 -31316.378,E2 -31316.378} C_VEL
LIN {X 0,Y 58.029,Z 353.595,A -85,B 0,C 180,E1 -31317.439,E2 -31317.439} C_VEL
LIN {X 0,Y 47.26,Z 362.439,A -85,B 0,C 180,E1 -31319.038,E2 -31319.038} C_VEL
LIN {X 0,Y 35.151,Z 370.597,A -85,B 0,C 180,E1 -31321.97,E2 -31321.97} C_VEL
LIN {X 0,Y 24.751,Z 376.406,A -85,B 0,C 180,E1 -31326.577,E2 -31326.577} C_VEL
LIN {X 0,Y 14.698,Z 381.106,A -85,B 0,C 180,E1 -31337.136,E2 -31337.136} C_VEL
LIN {X 0,Y 6.58,Z 384.865,A -85,B 0,C 180,E1 -31377.825,E2 -31377.825} C_VEL
LIN {X 0,Y 5.841,Z 385.93,A -85,B 0,C 180,E1 -31410.098,E2 -31410.098} C_VEL
LIN {X 0,Y 8.871,Z 387.694,A -85,B 0,C 180,E1 -31462.497,E2 -31462.497} C_VEL
LIN {X 0,Y 21.421,Z 390.151,A -85,B 0,C 180,E1 -31489.978,E2 -31489.978} C_VEL
LIN {X 0,Y 24.483,Z 390.467,A -85,B 0,C 180,E1 -31494.01,E2 -31494.01} C_VEL
LIN {X 0,Y 12.026,Z 388.274,A -85,B 0,C 180,E1 -31508.421,E2 -31508.421} C_VEL
LIN {X 0,Y 9.892,Z 390.227,A -85,B 0,C 180,E1 -31514.533,E2 -31514.533} C_VEL
LIN {X 0,Y 9.892,Z 600,A -85,B 0,C 180,E1 -31514.533,E2 -31514.533} C_VEL
LIN {X 0,Y 9.892,Z 600,A -85,B 0,C 180,E1 -31514.533,E2 -31514.533}

QRS_NEXT_CUT()

QRS_NEXT()
QRS_HOME()

END
